LIN {X 0,Y 573.039,Z 679.467,A -85,B 0,C 180,E1 -2242.601,E2 -2242.601} C_VEL
LIN {X 0,Y 573.014,Z 684.186,A -85,B 0,C 180,E1 -2244.016,E2 -2244.016} C_VEL
LIN {X 0,Y 573.006,Z 688.636,A -85,B 0,C 180,E1 -2245.78,E2 -2245.78} C_VEL
LIN {X 0,Y 572.947,Z 691.089,A -85,B 0,C 180,E1 -2247.188,E2 -2247.188} C_VEL
LIN {X 0,Y 572.939,Z 692.479,A -85,B 0,C 180,E1 -2248.594,E2 -2248.594} C_VEL
LIN {X 0,Y 572.933,Z 693,A -85,B 0,C 180,E1 -2250,E2 -2250} C_VEL
LIN {X 0,Y 572.939,Z 692.479,A -85,B 0,C 180,E1 -2251.406,E2 -2251.406} C_VEL
LIN {X 0,Y 572.947,Z 691.088,A -85,B 0,C 180,E1 -2252.812,E2 -2252.812} C_VEL
LIN {X 0,Y 573.006,Z 688.635,A -85,B 0,C 180,E1 -2254.22,E2 -2254.22} C_VEL
LIN {X 0,Y 573.013,Z 684.187,A -85,B 0,C 180,E1 -2255.984,E2 -2255.984} C_VEL
LIN {X 0,Y 573.04,Z 679.468,A -85,B 0,C 180,E1 -2257.399,E2 -2257.399} C_VEL
LIN {X 0,Y 573.076,Z 673.488,A -85,B 0,C 180,E1 -2258.818,E2 -2258.818} C_VEL
LIN {X 0,Y 573.182,Z 665.275,A -85,B 0,C 180,E1 -2260.42,E2 -2260.42} C_VEL
LIN {X 0,Y 573.269,Z 656.443,A -85,B 0,C 180,E1 -2261.85,E2 -2261.85} C_VEL
LIN {X 0,Y 573.448,Z 645.907,A -85,B 0,C 180,E1 -2263.285,E2 -2263.285} C_VEL
LIN {X 0,Y 573.59,Z 635.033,A -85,B 0,C 180,E1 -2264.544,E2 -2264.544} C_VEL
LIN {X 0,Y 573.831,Z 624.069,A -85,B 0,C 180,E1 -2265.631,E2 -2265.631} C_VEL
LIN {X 0,Y 574.091,Z 610.219,A -85,B 0,C 180,E1 -2266.811,E2 -2266.811} C_VEL
LIN {X 0,Y 574.357,Z 596.263,A -85,B 0,C 180,E1 -2267.813,E2 -2267.813} C_VEL
LIN {X 0,Y 574.633,Z 582.712,A -85,B 0,C 180,E1 -2268.634,E2 -2268.634} C_VEL
LIN {X 0,Y 574.868,Z 568.146,A -85,B 0,C 180,E1 -2269.364,E2 -2269.364} C_VEL
LIN {X 0,Y 575.126,Z 552.237,A -85,B 0,C 180,E1 -2270.009,E2 -2270.009} C_VEL
LIN {X 0,Y 575.36,Z 536.004,A -85,B 0,C 180,E1 -2270.513,E2 -2270.513} C_VEL
LIN {X 0,Y 575.491,Z 519.421,A -85,B 0,C 180,E1 -2270.882,E2 -2270.882} C_VEL
LIN {X 0,Y 576.17,Z 335.886,A -85,B 0,C 180,E1 -2273.297,E2 -2273.297} C_VEL
LIN {X 0,Y 576.126,Z 317.819,A -85,B 0,C 180,E1 -2273.539,E2 -2273.539} C_VEL
LIN {X 0,Y 575.046,Z 311.756,A -85,B 0,C 180,E1 -2273.688,E2 -2273.688} C_VEL
LIN {X 0,Y 575.605,Z 275.985,A -85,B 0,C 180,E1 -2276.796,E2 -2276.796} C_VEL
LIN {X 0,Y 575.436,Z 270.86,A -85,B 0,C 180,E1 -2277.258,E2 -2277.258} C_VEL
LIN {X 0,Y 573.251,Z 263.391,A -85,B 0,C 180,E1 -2278.039,E2 -2278.039} C_VEL
LIN {X 0,Y 573.232,Z 263.394,A -85,B 0,C 180,E1 -2280.883,E2 -2280.883} C_VEL
LIN {X 0,Y 573.262,Z 263.391,A -85,B 0,C 180,E1 -2283.524,E2 -2283.524} C_VEL
LIN {X 0,Y 573.213,Z 263.391,A -85,B 0,C 180,E1 -2286.052,E2 -2286.052} C_VEL
LIN {X 0,Y 573.248,Z 263.39,A -85,B 0,C 180,E1 -2288.701,E2 -2288.701} C_VEL
LIN {X 0,Y 573.244,Z 263.388,A -85,B 0,C 180,E1 -2291.595,E2 -2291.595} C_VEL
LIN {X 0,Y 573.24,Z 263.388,A -85,B 0,C 180,E1 -2294.333,E2 -2294.333} C_VEL
LIN {X 0,Y 573.241,Z 263.391,A -85,B 0,C 180,E1 -2297.359,E2 -2297.359} C_VEL
LIN {X 0,Y 573.248,Z 263.387,A -85,B 0,C 180,E1 -2300.393,E2 -2300.393} C_VEL
LIN {X 0,Y 573.253,Z 263.393,A -85,B 0,C 180,E1 -2303.078,E2 -2303.078} C_VEL
LIN {X 0,Y 573.267,Z 263.383,A -85,B 0,C 180,E1 -2305.672,E2 -2305.672} C_VEL
LIN {X 0,Y 573.243,Z 263.386,A -85,B 0,C 180,E1 -2308.185,E2 -2308.185} C_VEL
LIN {X 0,Y 573.265,Z 263.39,A -85,B 0,C 180,E1 -2310.635,E2 -2310.635} C_VEL
LIN {X 0,Y 573.251,Z 263.392,A -85,B 0,C 180,E1 -2313.024,E2 -2313.024} C_VEL
LIN {X 0,Y 573.276,Z 263.383,A -85,B 0,C 180,E1 -2315.367,E2 -2315.367} C_VEL
LIN {X 0,Y 573.229,Z 263.39,A -85,B 0,C 180,E1 -2318.42,E2 -2318.42} C_VEL
LIN {X 0,Y 573.271,Z 263.392,A -85,B 0,C 180,E1 -2320.732,E2 -2320.732} C_VEL
LIN {X 0,Y 573.242,Z 263.383,A -85,B 0,C 180,E1 -2323.622,E2 -2323.622} C_VEL
LIN {X 0,Y 573.229,Z 263.396,A -85,B 0,C 180,E1 -2326.53,E2 -2326.53} C_VEL
LIN {X 0,Y 573.265,Z 263.387,A -85,B 0,C 180,E1 -2328.746,E2 -2328.746} C_VEL
LIN {X 0,Y 573.254,Z 263.385,A -85,B 0,C 180,E1 -2331.54,E2 -2331.54} C_VEL
LIN {X 0,Y 573.285,Z 263.388,A -85,B 0,C 180,E1 -2334.372,E2 -2334.372} C_VEL
LIN {X 0,Y 573.311,Z 263.379,A -85,B 0,C 180,E1 -2337.893,E2 -2337.893} C_VEL
LIN {X 0,Y 573.327,Z 263.379,A -85,B 0,C 180,E1 -2340.703,E2 -2340.703} C_VEL
LIN {X 0,Y 573.291,Z 263.383,A -85,B 0,C 180,E1 -2342.811,E2 -2342.811} C_VEL
LIN {X 0,Y 573.271,Z 263.384,A -85,B 0,C 180,E1 -2345.629,E2 -2345.629} C_VEL
LIN {X 0,Y 573.25,Z 263.392,A -85,B 0,C 180,E1 -2348.46,E2 -2348.46} C_VEL
LIN {X 0,Y 573.275,Z 263.382,A -85,B 0,C 180,E1 -2351.312,E2 -2351.312} C_VEL
LIN {X 0,Y 573.273,Z 263.389,A -85,B 0,C 180,E1 -2354.42,E2 -2354.42} C_VEL
LIN {X 0,Y 573.195,Z 263.392,A -85,B 0,C 180,E1 -2357.114,E2 -2357.114} C_VEL
LIN {X 0,Y 573.268,Z 263.38,A -85,B 0,C 180,E1 -2359.33,E2 -2359.33} C_VEL
LIN {X 0,Y 573.209,Z 263.396,A -85,B 0,C 180,E1 -2362.339,E2 -2362.339} C_VEL
LIN {X 0,Y 573.202,Z 263.393,A -85,B 0,C 180,E1 -2364.375,E2 -2364.375} C_VEL
LIN {X 0,Y 572.56,Z 263.474,A -85,B 0,C 180,E1 -2364.962,E2 -2364.962} C_VEL
LIN {X 0,Y 569.719,Z 263.832,A -85,B 0,C 180,E1 -2365.913,E2 -2365.913} C_VEL
LIN {X 0,Y 567.293,Z 264.131,A -85,B 0,C 180,E1 -2366.679,E2 -2366.679} C_VEL
LIN {X 0,Y 566.236,Z 264.26,A -85,B 0,C 180,E1 -2367.27,E2 -2367.27} C_VEL
LIN {X 0,Y 566.142,Z 264.271,A -85,B 0,C 180,E1 -2367.47,E2 -2367.47} C_VEL
LIN {X 0,Y 566.158,Z 264.271,A -85,B 0,C 180,E1 -2370.595,E2 -2370.595} C_VEL
LIN {X 0,Y 566.162,Z 264.269,A -85,B 0,C 180,E1 -2373.107,E2 -2373.107} C_VEL
LIN {X 0,Y 566.133,Z 264.277,A -85,B 0,C 180,E1 -2375.695,E2 -2375.695} C_VEL
LIN {X 0,Y 566.187,Z 264.267,A -85,B 0,C 180,E1 -2378.555,E2 -2378.555} C_VEL
LIN {X 0,Y 566.136,Z 264.272,A -85,B 0,C 180,E1 -2381.144,E2 -2381.144} C_VEL
LIN {X 0,Y 566.149,Z 264.278,A -85,B 0,C 180,E1 -2384.041,E2 -2384.041} C_VEL
LIN {X 0,Y 566.155,Z 264.271,A -85,B 0,C 180,E1 -2387.089,E2 -2387.089} C_VEL
LIN {X 0,Y 566.19,Z 264.272,A -85,B 0,C 180,E1 -2390.318,E2 -2390.318} C_VEL
LIN {X 0,Y 566.221,Z 264.448,A -85,B 0,C 180,E1 -2391.127,E2 -2391.127} C_VEL
LIN {X 0,Y 568.077,Z 271.603,A -85,B 0,C 180,E1 -2391.953,E2 -2391.953} C_VEL
LIN {X 0,Y 568.103,Z 283.142,A -85,B 0,C 180,E1 -2393.09,E2 -2393.09} C_VEL
LIN {X 0,Y 569.669,Z 290.812,A -85,B 0,C 180,E1 -2393.263,E2 -2393.263} C_VEL
LIN {X 0,Y 568.911,Z 488.882,A -85,B 0,C 180,E1 -2395.901,E2 -2395.901} C_VEL
LIN {X 0,Y 568.673,Z 505.398,A -85,B 0,C 180,E1 -2396.264,E2 -2396.264} C_VEL
LIN {X 0,Y 568.446,Z 520.462,A -85,B 0,C 180,E1 -2396.727,E2 -2396.727} C_VEL
LIN {X 0,Y 568.229,Z 534.795,A -85,B 0,C 180,E1 -2397.288,E2 -2397.288} C_VEL
LIN {X 0,Y 567.885,Z 550.466,A -85,B 0,C 180,E1 -2398.058,E2 -2398.058} C_VEL
LIN {X 0,Y 567.583,Z 565.698,A -85,B 0,C 180,E1 -2398.975,E2 -2398.975} C_VEL
LIN {X 0,Y 567.236,Z 579.436,A -85,B 0,C 180,E1 -2399.963,E2 -2399.963} C_VEL
LIN {X 0,Y 566.924,Z 592.685,A -85,B 0,C 180,E1 -2401.087,E2 -2401.087} C_VEL
LIN {X 0,Y 566.675,Z 604.723,A -85,B 0,C 180,E1 -2402.284,E2 -2402.284} C_VEL
LIN {X 0,Y 566.438,Z 616.523,A -85,B 0,C 180,E1 -2403.668,E2 -2403.668} C_VEL
LIN {X 0,Y 566.25,Z 626.398,A -85,B 0,C 180,E1 -2405.04,E2 -2405.04} C_VEL
LIN {X 0,Y 566.132,Z 634.748,A -85,B 0,C 180,E1 -2406.4,E2 -2406.4} C_VEL
LIN {X 0,Y 566.023,Z 641.81,A -85,B 0,C 180,E1 -2407.747,E2 -2407.747} C_VEL
LIN {X 0,Y 565.958,Z 648.363,A -85,B 0,C 180,E1 -2409.273,E2 -2409.273} C_VEL
LIN {X 0,Y 565.919,Z 653.355,A -85,B 0,C 180,E1 -2410.706,E2 -2410.706} C_VEL
LIN {X 0,Y 565.856,Z 656.694,A -85,B 0,C 180,E1 -2411.91,E2 -2411.91} C_VEL
LIN {X 0,Y 565.845,Z 659.849,A -85,B 0,C 180,E1 -2413.401,E2 -2413.401} C_VEL
LIN {X 0,Y 565.805,Z 661.86,A -85,B 0,C 180,E1 -2414.88,E2 -2414.88} C_VEL
LIN {X 0,Y 565.863,Z 662.853,A -85,B 0,C 180,E1 -2416.351,E2 -2416.351} C_VEL
LIN {X 0,Y 565.864,Z 662.837,A -85,B 0,C 180,E1 -2417.811,E2 -2417.811} C_VEL
LIN {X 0,Y 565.893,Z 661.802,A -85,B 0,C 180,E1 -2419.264,E2 -2419.264} C_VEL
LIN {X 0,Y 565.829,Z 659.82,A -85,B 0,C 180,E1 -2420.708,E2 -2420.708} C_VEL
LIN {X 0,Y 565.879,Z 656.772,A -85,B 0,C 180,E1 -2422.148,E2 -2422.148} C_VEL
LIN {X 0,Y 565.948,Z 652.76,A -85,B 0,C 180,E1 -2423.583,E2 -2423.583} C_VEL
LIN {X 0,Y 565.989,Z 646.166,A -85,B 0,C 180,E1 -2425.37,E2 -2425.37} C_VEL
LIN {X 0,Y 566.057,Z 639.533,A -85,B 0,C 180,E1 -2426.797,E2 -2426.797} C_VEL
LIN {X 0,Y 566.173,Z 630.559,A -85,B 0,C 180,E1 -2428.399,E2 -2428.399} C_VEL
LIN {X 0,Y 566.305,Z 621.025,A -85,B 0,C 180,E1 -2429.822,E2 -2429.822} C_VEL
LIN {X 0,Y 566.52,Z 609.741,A -85,B 0,C 180,E1 -2431.244,E2 -2431.244} C_VEL
LIN {X 0,Y 566.818,Z 598.124,A -85,B 0,C 180,E1 -2432.487,E2 -2432.487} C_VEL
LIN {X 0,Y 567.115,Z 585.432,A -85,B 0,C 180,E1 -2433.641,E2 -2433.641} C_VEL
LIN {X 0,Y 567.384,Z 571.676,A -85,B 0,C 180,E1 -2434.707,E2 -2434.707} C_VEL
LIN {X 0,Y 567.697,Z 556.622,A -85,B 0,C 180,E1 -2435.684,E2 -2435.684} C_VEL
LIN {X 0,Y 568.054,Z 541.711,A -85,B 0,C 180,E1 -2436.482,E2 -2436.482} C_VEL
LIN {X 0,Y 568.372,Z 526.427,A -85,B 0,C 180,E1 -2437.147,E2 -2437.147} C_VEL
LIN {X 0,Y 568.633,Z 509.883,A -85,B 0,C 180,E1 -2437.702,E2 -2437.702} C_VEL
LIN {X 0,Y 568.827,Z 493.69,A -85,B 0,C 180,E1 -2438.096,E2 -2438.096} C_VEL
LIN {X 0,Y 568.984,Z 472.324,A -85,B 0,C 180,E1 -2438.426,E2 -2438.426} C_VEL
LIN {X 0,Y 569.662,Z 291.209,A -85,B 0,C 180,E1 -2440.822,E2 -2440.822} C_VEL
LIN {X 0,Y 568.055,Z 282.844,A -85,B 0,C 180,E1 -2441.011,E2 -2441.011} C_VEL
LIN {X 0,Y 568.099,Z 271.56,A -85,B 0,C 180,E1 -2442.14,E2 -2442.14} C_VEL
LIN {X 0,Y 566.179,Z 264.273,A -85,B 0,C 180,E1 -2443.002,E2 -2443.002} C_VEL
LIN {X 0,Y 566.189,Z 264.268,A -85,B 0,C 180,E1 -2445.11,E2 -2445.11} C_VEL
LIN {X 0,Y 566.171,Z 264.275,A -85,B 0,C 180,E1 -2448.079,E2 -2448.079} C_VEL
LIN {X 0,Y 566.197,Z 264.273,A -85,B 0,C 180,E1 -2450.338,E2 -2450.338} C_VEL
LIN {X 0,Y 566.17,Z 264.269,A -85,B 0,C 180,E1 -2453.28,E2 -2453.28} C_VEL
LIN {X 0,Y 566.174,Z 264.27,A -85,B 0,C 180,E1 -2455.751,E2 -2455.751} C_VEL
LIN {X 0,Y 566.138,Z 264.282,A -85,B 0,C 180,E1 -2458.189,E2 -2458.189} C_VEL
LIN {X 0,Y 566.176,Z 264.267,A -85,B 0,C 180,E1 -2461.073,E2 -2461.073} C_VEL
LIN {X 0,Y 566.184,Z 264.274,A -85,B 0,C 180,E1 -2463.958,E2 -2463.958} C_VEL
LIN {X 0,Y 566.122,Z 264.276,A -85,B 0,C 180,E1 -2466.576,E2 -2466.576} C_VEL
LIN {X 0,Y 566.179,Z 264.27,A -85,B 0,C 180,E1 -2469.681,E2 -2469.681} C_VEL
LIN {X 0,Y 566.144,Z 264.27,A -85,B 0,C 180,E1 -2472.91,E2 -2472.91} C_VEL
LIN {X 0,Y 566.146,Z 264.278,A -85,B 0,C 180,E1 -2475.959,E2 -2475.959} C_VEL
LIN {X 0,Y 566.135,Z 264.272,A -85,B 0,C 180,E1 -2478.856,E2 -2478.856} C_VEL
LIN {X 0,Y 566.174,Z 264.271,A -85,B 0,C 180,E1 -2481.635,E2 -2481.635} C_VEL
LIN {X 0,Y 566.136,Z 264.27,A -85,B 0,C 180,E1 -2484.305,E2 -2484.305} C_VEL
LIN {X 0,Y 566.164,Z 264.267,A -85,B 0,C 180,E1 -2486.894,E2 -2486.894} C_VEL
LIN {X 0,Y 566.168,Z 264.272,A -85,B 0,C 180,E1 -2489.406,E2 -2489.406} C_VEL
LIN {X 0,Y 566.144,Z 264.279,A -85,B 0,C 180,E1 -2491.853,E2 -2491.853} C_VEL
LIN {X 0,Y 566.185,Z 264.267,A -85,B 0,C 180,E1 -2494.249,E2 -2494.249} C_VEL
LIN {X 0,Y 566.168,Z 264.265,A -85,B 0,C 180,E1 -2496.72,E2 -2496.72} C_VEL
LIN {X 0,Y 566.204,Z 264.273,A -85,B 0,C 180,E1 -2499.662,E2 -2499.662} C_VEL
LIN {X 0,Y 566.18,Z 264.269,A -85,B 0,C 180,E1 -2501.921,E2 -2501.921} C_VEL
LIN {X 0,Y 566.19,Z 264.266,A -85,B 0,C 180,E1 -2504.89,E2 -2504.89} C_VEL
LIN {X 0,Y 566.217,Z 264.265,A -85,B 0,C 180,E1 -2507.818,E2 -2507.818} C_VEL
LIN {X 0,Y 566.17,Z 264.27,A -85,B 0,C 180,E1 -2509.992,E2 -2509.992} C_VEL
LIN {X 0,Y 566.237,Z 264.26,A -85,B 0,C 180,E1 -2512.87,E2 -2512.87} C_VEL
LIN {X 0,Y 566.274,Z 264.255,A -85,B 0,C 180,E1 -2515.016,E2 -2515.016} C_VEL
LIN {X 0,Y 566.284,Z 264.256,A -85,B 0,C 180,E1 -2517.866,E2 -2517.866} C_VEL
LIN {X 0,Y 566.292,Z 264.25,A -85,B 0,C 180,E1 -2520.711,E2 -2520.711} C_VEL
LIN {X 0,Y 566.263,Z 264.258,A -85,B 0,C 180,E1 -2522.845,E2 -2522.845} C_VEL
LIN {X 0,Y 566.263,Z 264.257,A -85,B 0,C 180,E1 -2525.698,E2 -2525.698} C_VEL
LIN {X 0,Y 566.226,Z 264.259,A -85,B 0,C 180,E1 -2528.565,E2 -2528.565} C_VEL
LIN {X 0,Y 566.243,Z 264.265,A -85,B 0,C 180,E1 -2531.454,E2 -2531.454} C_VEL
LIN {X 0,Y 566.224,Z 264.262,A -85,B 0,C 180,E1 -2534.502,E2 -2534.502} C_VEL
LIN {X 0,Y 566.2,Z 264.272,A -85,B 0,C 180,E1 -2537.331,E2 -2537.331} C_VEL
LIN {X 0,Y 566.207,Z 264.263,A -85,B 0,C 180,E1 -2540.337,E2 -2540.337} C_VEL
LIN {X 0,Y 566.19,Z 264.271,A -85,B 0,C 180,E1 -2543.403,E2 -2543.403} C_VEL
LIN {X 0,Y 566.213,Z 264.264,A -85,B 0,C 180,E1 -2545.749,E2 -2545.749} C_VEL
LIN {X 0,Y 566.202,Z 264.263,A -85,B 0,C 180,E1 -2548.202,E2 -2548.202} C_VEL
LIN {X 0,Y 566.191,Z 264.274,A -85,B 0,C 180,E1 -2551.076,E2 -2551.076} C_VEL
LIN {X 0,Y 566.211,Z 264.263,A -85,B 0,C 180,E1 -2553.734,E2 -2553.734} C_VEL
LIN {X 0,Y 566.209,Z 264.265,A -85,B 0,C 180,E1 -2556.569,E2 -2556.569} C_VEL
LIN {X 0,Y 566.212,Z 264.263,A -85,B 0,C 180,E1 -2559.685,E2 -2559.685} C_VEL
LIN {X 0,Y 566.21,Z 264.263,A -85,B 0,C 180,E1 -2562.087,E2 -2562.087} C_VEL
LIN {X 0,Y 566.173,Z 264.275,A -85,B 0,C 180,E1 -2565.036,E2 -2565.036} C_VEL
LIN {X 0,Y 566.217,Z 264.262,A -85,B 0,C 180,E1 -2568.136,E2 -2568.136} C_VEL
LIN {X 0,Y 566.22,Z 264.271,A -85,B 0,C 180,E1 -2570.727,E2 -2570.727} C_VEL
LIN {X 0,Y 566.184,Z 264.266,A -85,B 0,C 180,E1 -2573.788,E2 -2573.788} C_VEL
LIN {X 0,Y 566.21,Z 264.266,A -85,B 0,C 180,E1 -2576.266,E2 -2576.266} C_VEL
LIN {X 0,Y 566.192,Z 264.273,A -85,B 0,C 180,E1 -2578.923,E2 -2578.923} C_VEL
LIN {X 0,Y 566.241,Z 264.43,A -85,B 0,C 180,E1 -2581.703,E2 -2581.703} C_VEL
LIN {X 0,Y 568.802,Z 273.142,A -85,B 0,C 180,E1 -2582.617,E2 -2582.617} C_VEL
LIN {X 0,Y 568.734,Z 288.517,A -85,B 0,C 180,E1 -2583.98,E2 -2583.98} C_VEL
LIN {X 0,Y 568.339,Z 311.989,A -85,B 0,C 180,E1 -2586.035,E2 -2586.035} C_VEL
LIN {X 0,Y 569.734,Z 319.826,A -85,B 0,C 180,E1 -2586.208,E2 -2586.208} C_VEL
LIN {X 0,Y 568.878,Z 519.43,A -85,B 0,C 180,E1 -2588.864,E2 -2588.864} C_VEL
LIN {X 0,Y 568.726,Z 536.008,A -85,B 0,C 180,E1 -2589.237,E2 -2589.237} C_VEL
LIN {X 0,Y 568.422,Z 552.242,A -85,B 0,C 180,E1 -2589.745,E2 -2589.745} C_VEL
LIN {X 0,Y 568.145,Z 568.386,A -85,B 0,C 180,E1 -2590.408,E2 -2590.408} C_VEL
LIN {X 0,Y 567.878,Z 582.716,A -85,B 0,C 180,E1 -2591.136,E2 -2591.136} C_VEL
LIN {X 0,Y 567.582,Z 596.269,A -85,B 0,C 180,E1 -2591.967,E2 -2591.967} C_VEL
LIN {X 0,Y 567.228,Z 610.219,A -85,B 0,C 180,E1 -2592.979,E2 -2592.979} C_VEL
LIN {X 0,Y 566.915,Z 624.07,A -85,B 0,C 180,E1 -2594.173,E2 -2594.173} C_VEL
LIN {X 0,Y 566.63,Z 635.619,A -85,B 0,C 180,E1 -2595.339,E2 -2595.339} C_VEL
LIN {X 0,Y 566.434,Z 647.337,A -85,B 0,C 180,E1 -2596.73,E2 -2596.73} C_VEL
LIN {X 0,Y 566.238,Z 657.673,A -85,B 0,C 180,E1 -2598.183,E2 -2598.183} C_VEL
LIN {X 0,Y 566.12,Z 666.284,A -85,B 0,C 180,E1 -2599.63,E2 -2599.63} C_VEL
LIN {X 0,Y 566.001,Z 673.489,A -85,B 0,C 180,E1 -2601.071,E2 -2601.071} C_VEL
LIN {X 0,Y 565.968,Z 679.467,A -85,B 0,C 180,E1 -2602.508,E2 -2602.508} C_VEL
LIN {X 0,Y 565.915,Z 684.187,A -85,B 0,C 180,E1 -2603.941,E2 -2603.941} C_VEL
LIN {X 0,Y 565.911,Z 688.637,A -85,B 0,C 180,E1 -2605.727,E2 -2605.727} C_VEL
LIN {X 0,Y 565.865,Z 691.089,A -85,B 0,C 180,E1 -2607.152,E2 -2607.152} C_VEL
LIN {X 0,Y 565.839,Z 692.48,A -85,B 0,C 180,E1 -2608.577,E2 -2608.577} C_VEL
LIN {X 0,Y 565.834,Z 693,A -85,B 0,C 180,E1 -2610,E2 -2610} C_VEL
LIN {X 0,Y 565.839,Z 692.48,A -85,B 0,C 180,E1 -2611.424,E2 -2611.424} C_VEL
LIN {X 0,Y 565.866,Z 691.088,A -85,B 0,C 180,E1 -2612.848,E2 -2612.848} C_VEL
LIN {X 0,Y 565.911,Z 688.636,A -85,B 0,C 180,E1 -2614.273,E2 -2614.273} C_VEL
LIN {X 0,Y 565.914,Z 684.188,A -85,B 0,C 180,E1 -2616.06,E2 -2616.06} C_VEL
LIN {X 0,Y 565.968,Z 679.468,A -85,B 0,C 180,E1 -2617.492,E2 -2617.492} C_VEL
LIN {X 0,Y 566.001,Z 673.489,A -85,B 0,C 180,E1 -2618.929,E2 -2618.929} C_VEL
LIN {X 0,Y 566.126,Z 665.276,A -85,B 0,C 180,E1 -2620.551,E2 -2620.551} C_VEL
LIN {X 0,Y 566.246,Z 656.442,A -85,B 0,C 180,E1 -2621.999,E2 -2621.999} C_VEL
LIN {X 0,Y 566.427,Z 645.907,A -85,B 0,C 180,E1 -2623.453,E2 -2623.453} C_VEL
LIN {X 0,Y 566.661,Z 634.61,A -85,B 0,C 180,E1 -2624.774,E2 -2624.774} C_VEL
LIN {X 0,Y 566.958,Z 622.117,A -85,B 0,C 180,E1 -2626.01,E2 -2626.01} C_VEL
LIN {X 0,Y 567.229,Z 609.043,A -85,B 0,C 180,E1 -2627.113,E2 -2627.113} C_VEL
LIN {X 0,Y 567.581,Z 594.848,A -85,B 0,C 180,E1 -2628.126,E2 -2628.126} C_VEL
LIN {X 0,Y 567.907,Z 579.276,A -85,B 0,C 180,E1 -2629.05,E2 -2629.05} C_VEL
LIN {X 0,Y 568.272,Z 563.648,A -85,B 0,C 180,E1 -2629.804,E2 -2629.804} C_VEL
LIN {X 0,Y 568.551,Z 547.003,A -85,B 0,C 180,E1 -2630.439,E2 -2630.439} C_VEL
LIN {X 0,Y 568.778,Z 530.512,A -85,B 0,C 180,E1 -2630.903,E2 -2630.903} C_VEL
LIN {X 0,Y 568.899,Z 514.918,A -85,B 0,C 180,E1 -2631.207,E2 -2631.207} C_VEL
LIN {X 0,Y 569.679,Z 320,A -85,B 0,C 180,E1 -2633.792,E2 -2633.792} C_VEL
LIN {X 0,Y 568.354,Z 311.822,A -85,B 0,C 180,E1 -2633.979,E2 -2633.979} C_VEL
LIN {X 0,Y 568.944,Z 276.843,A -85,B 0,C 180,E1 -2637.044,E2 -2637.044} C_VEL
LIN {X 0,Y 568.742,Z 272.884,A -85,B 0,C 180,E1 -2637.406,E2 -2637.406} C_VEL
LIN {X 0,Y 566.216,Z 264.268,A -85,B 0,C 180,E1 -2638.324,E2 -2638.324} C_VEL
LIN {X 0,Y 566.195,Z 264.273,A -85,B 0,C 180,E1 -2641.422,E2 -2641.422} C_VEL
LIN {X 0,Y 566.209,Z 264.265,A -85,B 0,C 180,E1 -2643.956,E2 -2643.956} C_VEL
LIN {X 0,Y 566.199,Z 264.267,A -85,B 0,C 180,E1 -2646.57,E2 -2646.57} C_VEL
LIN {X 0,Y 566.221,Z 264.269,A -85,B 0,C 180,E1 -2649.273,E2 -2649.273} C_VEL
LIN {X 0,Y 566.211,Z 264.261,A -85,B 0,C 180,E1 -2652.088,E2 -2652.088} C_VEL
LIN {X 0,Y 566.174,Z 264.274,A -85,B 0,C 180,E1 -2655.036,E2 -2655.036} C_VEL
LIN {X 0,Y 566.218,Z 264.261,A -85,B 0,C 180,E1 -2658.136,E2 -2658.136} C_VEL
LIN {X 0,Y 566.223,Z 264.267,A -85,B 0,C 180,E1 -2660.727,E2 -2660.727} C_VEL
LIN {X 0,Y 566.185,Z 264.266,A -85,B 0,C 180,E1 -2663.788,E2 -2663.788} C_VEL
LIN {X 0,Y 566.212,Z 264.263,A -85,B 0,C 180,E1 -2666.266,E2 -2666.266} C_VEL
LIN {X 0,Y 566.194,Z 264.274,A -85,B 0,C 180,E1 -2668.924,E2 -2668.924} C_VEL
LIN {X 0,Y 566.213,Z 264.258,A -85,B 0,C 180,E1 -2671.858,E2 -2671.858} C_VEL
LIN {X 0,Y 566.214,Z 264.264,A -85,B 0,C 180,E1 -2674.251,E2 -2674.251} C_VEL
LIN {X 0,Y 566.174,Z 264.273,A -85,B 0,C 180,E1 -2676.719,E2 -2676.719} C_VEL
LIN {X 0,Y 566.207,Z 264.263,A -85,B 0,C 180,E1 -2679.663,E2 -2679.663} C_VEL
LIN {X 0,Y 566.201,Z 264.268,A -85,B 0,C 180,E1 -2682.669,E2 -2682.669} C_VEL
LIN {X 0,Y 566.223,Z 264.261,A -85,B 0,C 180,E1 -2685.627,E2 -2685.627} C_VEL
LIN {X 0,Y 566.237,Z 264.263,A -85,B 0,C 180,E1 -2688.676,E2 -2688.676} C_VEL
LIN {X 0,Y 566.205,Z 264.263,A -85,B 0,C 180,E1 -2691.434,E2 -2691.434} C_VEL
LIN {X 0,Y 566.253,Z 264.263,A -85,B 0,C 180,E1 -2694.302,E2 -2694.302} C_VEL
LIN {X 0,Y 566.282,Z 264.254,A -85,B 0,C 180,E1 -2697.867,E2 -2697.867} C_VEL
LIN {X 0,Y 566.298,Z 264.253,A -85,B 0,C 180,E1 -2700.711,E2 -2700.711} C_VEL
LIN {X 0,Y 566.257,Z 264.259,A -85,B 0,C 180,E1 -2702.846,E2 -2702.846} C_VEL
LIN {X 0,Y 566.241,Z 264.26,A -85,B 0,C 180,E1 -2705.699,E2 -2705.699} C_VEL
LIN {X 0,Y 566.201,Z 264.268,A -85,B 0,C 180,E1 -2708.567,E2 -2708.567} C_VEL
LIN {X 0,Y 566.243,Z 264.259,A -85,B 0,C 180,E1 -2711.455,E2 -2711.455} C_VEL
LIN {X 0,Y 566.227,Z 264.265,A -85,B 0,C 180,E1 -2714.502,E2 -2714.502} C_VEL
LIN {X 0,Y 566.161,Z 264.269,A -85,B 0,C 180,E1 -2717.333,E2 -2717.333} C_VEL
LIN {X 0,Y 566.199,Z 264.261,A -85,B 0,C 180,E1 -2719.581,E2 -2719.581} C_VEL
LIN {X 0,Y 566.179,Z 264.272,A -85,B 0,C 180,E1 -2721.864,E2 -2721.864} C_VEL
LIN {X 0,Y 566.15,Z 264.273,A -85,B 0,C 180,E1 -2724.372,E2 -2724.372} C_VEL
LIN {X 0,Y 566.16,Z 264.271,A -85,B 0,C 180,E1 -2726.649,E2 -2726.649} C_VEL
LIN {X 0,Y 566.142,Z 264.271,A -85,B 0,C 180,E1 -2727.47,E2 -2727.47} C_VEL
LIN {X 0,Y 565.452,Z 264.363,A -85,B 0,C 180,E1 -2728.064,E2 -2728.064} C_VEL
LIN {X 0,Y 562.584,Z 264.72,A -85,B 0,C 180,E1 -2729.028,E2 -2729.028} C_VEL
LIN {X 0,Y 560.187,Z 265.019,A -85,B 0,C 180,E1 -2729.803,E2 -2729.803} C_VEL
LIN {X 0,Y 559.177,Z 265.144,A -85,B 0,C 180,E1 -2730.402,E2 -2730.402} C_VEL
LIN {X 0,Y 559.105,Z 265.15,A -85,B 0,C 180,E1 -2730.605,E2 -2730.605} C_VEL
LIN {X 0,Y 559.134,Z 265.145,A -85,B 0,C 180,E1 -2732.717,E2 -2732.717} C_VEL
LIN {X 0,Y 559.111,Z 265.148,A -85,B 0,C 180,E1 -2735.326,E2 -2735.326} C_VEL
LIN {X 0,Y 559.108,Z 265.154,A -85,B 0,C 180,E1 -2738.02,E2 -2738.02} C_VEL
LIN {X 0,Y 559.093,Z 265.149,A -85,B 0,C 180,E1 -2740.819,E2 -2740.819} C_VEL
LIN {X 0,Y 559.095,Z 265.158,A -85,B 0,C 180,E1 -2743.739,E2 -2743.739} C_VEL
LIN {X 0,Y 559.103,Z 265.152,A -85,B 0,C 180,E1 -2746.262,E2 -2746.262} C_VEL
LIN {X 0,Y 559.098,Z 265.151,A -85,B 0,C 180,E1 -2748.958,E2 -2748.958} C_VEL
LIN {X 0,Y 559.192,Z 265.316,A -85,B 0,C 180,E1 -2750.847,E2 -2750.847} C_VEL
LIN {X 0,Y 561.485,Z 274.746,A -85,B 0,C 180,E1 -2751.943,E2 -2751.943} C_VEL
LIN {X 0,Y 561.415,Z 283.251,A -85,B 0,C 180,E1 -2752.786,E2 -2752.786} C_VEL
LIN {X 0,Y 563.161,Z 291.947,A -85,B 0,C 180,E1 -2752.986,E2 -2752.986} C_VEL
LIN {X 0,Y 562.3,Z 486.908,A -85,B 0,C 180,E1 -2755.609,E2 -2755.609} C_VEL
LIN {X 0,Y 562.049,Z 503.604,A -85,B 0,C 180,E1 -2755.961,E2 -2755.961} C_VEL
LIN {X 0,Y 561.792,Z 519.55,A -85,B 0,C 180,E1 -2756.442,E2 -2756.442} C_VEL
LIN {X 0,Y 561.511,Z 535.019,A -85,B 0,C 180,E1 -2757.051,E2 -2757.051} C_VEL
LIN {X 0,Y 561.106,Z 550.799,A -85,B 0,C 180,E1 -2757.837,E2 -2757.837} C_VEL
LIN {X 0,Y 560.784,Z 565.257,A -85,B 0,C 180,E1 -2758.719,E2 -2758.719} C_VEL
LIN {X 0,Y 560.394,Z 578.625,A -85,B 0,C 180,E1 -2759.683,E2 -2759.683} C_VEL
LIN {X 0,Y 560.049,Z 591.799,A -85,B 0,C 180,E1 -2760.801,E2 -2760.801} C_VEL
LIN {X 0,Y 559.724,Z 604.87,A -85,B 0,C 180,E1 -2762.114,E2 -2762.114} C_VEL
LIN {X 0,Y 559.444,Z 616.653,A -85,B 0,C 180,E1 -2763.515,E2 -2763.515} C_VEL
LIN {X 0,Y 559.231,Z 625.839,A -85,B 0,C 180,E1 -2764.803,E2 -2764.803} C_VEL
LIN {X 0,Y 559.07,Z 634.839,A -85,B 0,C 180,E1 -2766.28,E2 -2766.28} C_VEL
LIN {X 0,Y 558.93,Z 642.764,A -85,B 0,C 180,E1 -2767.838,E2 -2767.838} C_VEL
LIN {X 0,Y 558.857,Z 649.181,A -85,B 0,C 180,E1 -2769.383,E2 -2769.383} C_VEL
LIN {X 0,Y 558.814,Z 654.204,A -85,B 0,C 180,E1 -2770.914,E2 -2770.914} C_VEL
LIN {X 0,Y 558.756,Z 658.059,A -85,B 0,C 180,E1 -2772.43,E2 -2772.43} C_VEL
LIN {X 0,Y 558.728,Z 660.745,A -85,B 0,C 180,E1 -2773.935,E2 -2773.935} C_VEL
LIN {X 0,Y 558.763,Z 662.464,A -85,B 0,C 180,E1 -2775.58,E2 -2775.58} C_VEL
LIN {X 0,Y 558.741,Z 662.978,A -85,B 0,C 180,E1 -2776.914,E2 -2776.914} C_VEL
LIN {X 0,Y 558.801,Z 662.261,A -85,B 0,C 180,E1 -2778.816,E2 -2778.816} C_VEL
LIN {X 0,Y 558.778,Z 661.178,A -85,B 0,C 180,E1 -2779.858,E2 -2779.858} C_VEL
LIN {X 0,Y 558.766,Z 658.745,A -85,B 0,C 180,E1 -2781.319,E2 -2781.319} C_VEL
LIN {X 0,Y 558.804,Z 655.375,A -85,B 0,C 180,E1 -2782.775,E2 -2782.775} C_VEL
LIN {X 0,Y 558.87,Z 649.627,A -85,B 0,C 180,E1 -2784.588,E2 -2784.588} C_VEL
LIN {X 0,Y 558.954,Z 643.725,A -85,B 0,C 180,E1 -2786.035,E2 -2786.035} C_VEL
LIN {X 0,Y 559.022,Z 636.671,A -85,B 0,C 180,E1 -2787.478,E2 -2787.478} C_VEL
LIN {X 0,Y 559.198,Z 628.262,A -85,B 0,C 180,E1 -2788.92,E2 -2788.92} C_VEL
LIN {X 0,Y 559.336,Z 618.269,A -85,B 0,C 180,E1 -2790.36,E2 -2790.36} C_VEL
LIN {X 0,Y 559.601,Z 608.024,A -85,B 0,C 180,E1 -2791.619,E2 -2791.619} C_VEL
LIN {X 0,Y 559.941,Z 596.116,A -85,B 0,C 180,E1 -2792.878,E2 -2792.878} C_VEL
LIN {X 0,Y 560.32,Z 583.146,A -85,B 0,C 180,E1 -2794.046,E2 -2794.046} C_VEL
LIN {X 0,Y 560.596,Z 571.449,A -85,B 0,C 180,E1 -2794.944,E2 -2794.944} C_VEL
LIN {X 0,Y 560.876,Z 557.881,A -85,B 0,C 180,E1 -2795.843,E2 -2795.843} C_VEL
LIN {X 0,Y 561.289,Z 543.266,A -85,B 0,C 180,E1 -2796.651,E2 -2796.651} C_VEL
LIN {X 0,Y 561.657,Z 527.124,A -85,B 0,C 180,E1 -2797.369,E2 -2797.369} C_VEL
LIN {X 0,Y 561.961,Z 511.524,A -85,B 0,C 180,E1 -2797.907,E2 -2797.907} C_VEL
LIN {X 0,Y 562.215,Z 495.019,A -85,B 0,C 180,E1 -2798.328,E2 -2798.328} C_VEL
LIN {X 0,Y 562.362,Z 477.198,A -85,B 0,C 180,E1 -2798.625,E2 -2798.625} C_VEL
LIN {X 0,Y 563.153,Z 291.665,A -85,B 0,C 180,E1 -2801.108,E2 -2801.108} C_VEL
LIN {X 0,Y 561.326,Z 282.817,A -85,B 0,C 180,E1 -2801.327,E2 -2801.327} C_VEL
LIN {X 0,Y 561.356,Z 273.43,A -85,B 0,C 180,E1 -2802.288,E2 -2802.288} C_VEL
LIN {X 0,Y 559.162,Z 265.147,A -85,B 0,C 180,E1 -2803.284,E2 -2803.284} C_VEL
LIN {X 0,Y 559.137,Z 265.147,A -85,B 0,C 180,E1 -2805.305,E2 -2805.305} C_VEL
LIN {X 0,Y 559.125,Z 265.147,A -85,B 0,C 180,E1 -2807.558,E2 -2807.558} C_VEL
LIN {X 0,Y 559.164,Z 265.145,A -85,B 0,C 180,E1 -2809.838,E2 -2809.838} C_VEL
LIN {X 0,Y 559.132,Z 265.15,A -85,B 0,C 180,E1 -2812.153,E2 -2812.153} C_VEL
LIN {X 0,Y 559.141,Z 265.143,A -85,B 0,C 180,E1 -2815.177,E2 -2815.177} C_VEL
LIN {X 0,Y 559.098,Z 265.152,A -85,B 0,C 180,E1 -2817.717,E2 -2817.717} C_VEL
LIN {X 0,Y 559.13,Z 265.155,A -85,B 0,C 180,E1 -2820.184,E2 -2820.184} C_VEL
LIN {X 0,Y 559.135,Z 265.146,A -85,B 0,C 180,E1 -2822.717,E2 -2822.717} C_VEL
LIN {X 0,Y 559.112,Z 265.146,A -85,B 0,C 180,E1 -2825.325,E2 -2825.325} C_VEL
LIN {X 0,Y 559.085,Z 265.158,A -85,B 0,C 180,E1 -2828.021,E2 -2828.021} C_VEL
LIN {X 0,Y 559.119,Z 265.154,A -85,B 0,C 180,E1 -2829.936,E2 -2829.936} C_VEL
LIN {X 0,Y 559.108,Z 265.147,A -85,B 0,C 180,E1 -2832.748,E2 -2832.748} C_VEL
LIN {X 0,Y 559.114,Z 265.153,A -85,B 0,C 180,E1 -2835.765,E2 -2835.765} C_VEL
LIN {X 0,Y 559.095,Z 265.154,A -85,B 0,C 180,E1 -2838.223,E2 -2838.223} C_VEL
LIN {X 0,Y 559.168,Z 265.139,A -85,B 0,C 180,E1 -2841.193,E2 -2841.193} C_VEL
LIN {X 0,Y 559.108,Z 265.146,A -85,B 0,C 180,E1 -2843.786,E2 -2843.786} C_VEL
LIN {X 0,Y 559.138,Z 265.144,A -85,B 0,C 180,E1 -2846.423,E2 -2846.423} C_VEL
LIN {X 0,Y 559.149,Z 265.142,A -85,B 0,C 180,E1 -2848.98,E2 -2848.98} C_VEL
LIN {X 0,Y 559.105,Z 265.152,A -85,B 0,C 180,E1 -2851.631,E2 -2851.631} C_VEL
LIN {X 0,Y 559.126,Z 265.144,A -85,B 0,C 180,E1 -2854.699,E2 -2854.699} C_VEL
LIN {X 0,Y 559.119,Z 265.145,A -85,B 0,C 180,E1 -2857.066,E2 -2857.066} C_VEL
LIN {X 0,Y 559.175,Z 265.144,A -85,B 0,C 180,E1 -2859.395,E2 -2859.395} C_VEL
LIN {X 0,Y 559.129,Z 265.15,A -85,B 0,C 180,E1 -2861.685,E2 -2861.685} C_VEL
LIN {X 0,Y 559.145,Z 265.147,A -85,B 0,C 180,E1 -2863.947,E2 -2863.947} C_VEL
LIN {X 0,Y 559.16,Z 265.142,A -85,B 0,C 180,E1 -2866.183,E2 -2866.183} C_VEL
LIN {X 0,Y 559.193,Z 265.137,A -85,B 0,C 180,E1 -2869.133,E2 -2869.133} C_VEL
LIN {X 0,Y 559.173,Z 265.141,A -85,B 0,C 180,E1 -2872.053,E2 -2872.053} C_VEL
LIN {X 0,Y 559.248,Z 265.129,A -85,B 0,C 180,E1 -2874.953,E2 -2874.953} C_VEL
LIN {X 0,Y 559.255,Z 265.132,A -85,B 0,C 180,E1 -2877.839,E2 -2877.839} C_VEL
LIN {X 0,Y 559.264,Z 265.125,A -85,B 0,C 180,E1 -2880.72,E2 -2880.72} C_VEL
LIN {X 0,Y 559.231,Z 265.134,A -85,B 0,C 180,E1 -2882.881,E2 -2882.881} C_VEL
LIN {X 0,Y 559.231,Z 265.132,A -85,B 0,C 180,E1 -2885.77,E2 -2885.77} C_VEL
LIN {X 0,Y 559.185,Z 265.137,A -85,B 0,C 180,E1 -2888.674,E2 -2888.674} C_VEL
LIN {X 0,Y 559.206,Z 265.139,A -85,B 0,C 180,E1 -2891.6,E2 -2891.6} C_VEL
LIN {X 0,Y 559.181,Z 265.14,A -85,B 0,C 180,E1 -2894.587,E2 -2894.587} C_VEL
LIN {X 0,Y 559.143,Z 265.147,A -85,B 0,C 180,E1 -2897.557,E2 -2897.557} C_VEL
LIN {X 0,Y 559.166,Z 265.142,A -85,B 0,C 180,E1 -2899.837,E2 -2899.837} C_VEL
LIN {X 0,Y 559.141,Z 265.143,A -85,B 0,C 180,E1 -2902.152,E2 -2902.152} C_VEL
LIN {X 0,Y 559.179,Z 265.147,A -85,B 0,C 180,E1 -2905.187,E2 -2905.187} C_VEL
LIN {X 0,Y 559.157,Z 265.142,A -85,B 0,C 180,E1 -2907.713,E2 -2907.713} C_VEL
LIN {X 0,Y 559.153,Z 265.142,A -85,B 0,C 180,E1 -2910.182,E2 -2910.182} C_VEL
LIN {X 0,Y 559.156,Z 265.147,A -85,B 0,C 180,E1 -2912.715,E2 -2912.715} C_VEL
LIN {X 0,Y 559.144,Z 265.146,A -85,B 0,C 180,E1 -2915.322,E2 -2915.322} C_VEL
LIN {X 0,Y 559.135,Z 265.144,A -85,B 0,C 180,E1 -2918.017,E2 -2918.017} C_VEL
LIN {X 0,Y 559.175,Z 265.146,A -85,B 0,C 180,E1 -2920.81,E2 -2920.81} C_VEL
LIN {X 0,Y 559.14,Z 265.143,A -85,B 0,C 180,E1 -2923.734,E2 -2923.734} C_VEL
LIN {X 0,Y 559.167,Z 265.149,A -85,B 0,C 180,E1 -2926.801,E2 -2926.801} C_VEL
LIN {X 0,Y 559.176,Z 265.144,A -85,B 0,C 180,E1 -2929.189,E2 -2929.189} C_VEL
LIN {X 0,Y 559.133,Z 265.145,A -85,B 0,C 180,E1 -2931.982,E2 -2931.982} C_VEL
LIN {X 0,Y 559.13,Z 265.152,A -85,B 0,C 180,E1 -2934.787,E2 -2934.787} C_VEL
LIN {X 0,Y 559.154,Z 265.145,A -85,B 0,C 180,E1 -2937.364,E2 -2937.364} C_VEL
LIN {X 0,Y 559.146,Z 265.148,A -85,B 0,C 180,E1 -2940.143,E2 -2940.143} C_VEL
LIN {X 0,Y 559.196,Z 265.258,A -85,B 0,C 180,E1 -2941.408,E2 -2941.408} C_VEL
LIN {X 0,Y 562.249,Z 276.142,A -85,B 0,C 180,E1 -2942.558,E2 -2942.558} C_VEL
LIN {X 0,Y 561.812,Z 301.706,A -85,B 0,C 180,E1 -2944.829,E2 -2944.829} C_VEL
LIN {X 0,Y 561.68,Z 312.356,A -85,B 0,C 180,E1 -2945.743,E2 -2945.743} C_VEL
LIN {X 0,Y 563.221,Z 321.181,A -85,B 0,C 180,E1 -2945.934,E2 -2945.934} C_VEL
LIN {X 0,Y 562.293,Z 517.938,A -85,B 0,C 180,E1 -2948.58,E2 -2948.58} C_VEL
LIN {X 0,Y 562.073,Z 534.177,A -85,B 0,C 180,E1 -2948.932,E2 -2948.932} C_VEL
LIN {X 0,Y 561.787,Z 550.94,A -85,B 0,C 180,E1 -2949.448,E2 -2949.448} C_VEL
LIN {X 0,Y 561.501,Z 565.854,A -85,B 0,C 180,E1 -2950.045,E2 -2950.045} C_VEL
LIN {X 0,Y 561.137,Z 581.034,A -85,B 0,C 180,E1 -2950.806,E2 -2950.806} C_VEL
LIN {X 0,Y 560.779,Z 594.849,A -85,B 0,C 180,E1 -2951.646,E2 -2951.646} C_VEL
LIN {X 0,Y 560.367,Z 609.043,A -85,B 0,C 180,E1 -2952.671,E2 -2952.671} C_VEL
LIN {X 0,Y 559.988,Z 622.118,A -85,B 0,C 180,E1 -2953.785,E2 -2953.785} C_VEL
LIN {X 0,Y 559.722,Z 634.654,A -85,B 0,C 180,E1 -2955.044,E2 -2955.044} C_VEL
LIN {X 0,Y 559.448,Z 645.907,A -85,B 0,C 180,E1 -2956.376,E2 -2956.376} C_VEL
LIN {X 0,Y 559.219,Z 656.441,A -85,B 0,C 180,E1 -2957.848,E2 -2957.848} C_VEL
LIN {X 0,Y 559.057,Z 665.276,A -85,B 0,C 180,E1 -2959.314,E2 -2959.314} C_VEL
LIN {X 0,Y 558.93,Z 671.856,A -85,B 0,C 180,E1 -2960.592,E2 -2960.592} C_VEL
LIN {X 0,Y 558.893,Z 679.466,A -85,B 0,C 180,E1 -2962.413,E2 -2962.413} C_VEL
LIN {X 0,Y 558.863,Z 685.248,A -85,B 0,C 180,E1 -2964.226,E2 -2964.226} C_VEL
LIN {X 0,Y 558.805,Z 688.636,A -85,B 0,C 180,E1 -2965.672,E2 -2965.672} C_VEL
LIN {X 0,Y 558.787,Z 691.09,A -85,B 0,C 180,E1 -2967.116,E2 -2967.116} C_VEL
LIN {X 0,Y 558.739,Z 692.48,A -85,B 0,C 180,E1 -2968.559,E2 -2968.559} C_VEL
LIN {X 0,Y 558.735,Z 693,A -85,B 0,C 180,E1 -2970,E2 -2970} C_VEL
LIN {X 0,Y 558.738,Z 692.479,A -85,B 0,C 180,E1 -2971.442,E2 -2971.442} C_VEL
LIN {X 0,Y 558.787,Z 691.088,A -85,B 0,C 180,E1 -2972.884,E2 -2972.884} C_VEL
LIN {X 0,Y 558.805,Z 688.635,A -85,B 0,C 180,E1 -2974.328,E2 -2974.328} C_VEL
LIN {X 0,Y 558.862,Z 685.249,A -85,B 0,C 180,E1 -2975.774,E2 -2975.774} C_VEL
LIN {X 0,Y 558.893,Z 679.467,A -85,B 0,C 180,E1 -2977.587,E2 -2977.587} C_VEL
LIN {X 0,Y 558.93,Z 671.856,A -85,B 0,C 180,E1 -2979.408,E2 -2979.408} C_VEL
LIN {X 0,Y 559.116,Z 663.28,A -85,B 0,C 180,E1 -2981.046,E2 -2981.046} C_VEL
LIN {X 0,Y 559.275,Z 653.975,A -85,B 0,C 180,E1 -2982.519,E2 -2982.519} C_VEL
LIN {X 0,Y 559.471,Z 644.421,A -85,B 0,C 180,E1 -2983.808,E2 -2983.808} C_VEL
LIN {X 0,Y 559.791,Z 633.258,A -85,B 0,C 180,E1 -2985.103,E2 -2985.103} C_VEL
LIN {X 0,Y 560.05,Z 621.139,A -85,B 0,C 180,E1 -2986.307,E2 -2986.307} C_VEL
LIN {X 0,Y 560.42,Z 607.868,A -85,B 0,C 180,E1 -2987.422,E2 -2987.422} C_VEL
LIN {X 0,Y 560.786,Z 594.845,A -85,B 0,C 180,E1 -2988.353,E2 -2988.353} C_VEL
LIN {X 0,Y 561.133,Z 581.026,A -85,B 0,C 180,E1 -2989.194,E2 -2989.194} C_VEL
LIN {X 0,Y 561.469,Z 566.936,A -85,B 0,C 180,E1 -2989.904,E2 -2989.904} C_VEL
LIN {X 0,Y 561.773,Z 550.936,A -85,B 0,C 180,E1 -2990.553,E2 -2990.553} C_VEL
LIN {X 0,Y 562.11,Z 534.176,A -85,B 0,C 180,E1 -2991.067,E2 -2991.067} C_VEL
LIN {X 0,Y 562.273,Z 517.929,A -85,B 0,C 180,E1 -2991.421,E2 -2991.421} C_VEL
LIN {X 0,Y 563.202,Z 320.984,A -85,B 0,C 180,E1 -2994.07,E2 -2994.07} C_VEL
LIN {X 0,Y 561.619,Z 311.974,A -85,B 0,C 180,E1 -2994.27,E2 -2994.27} C_VEL
LIN {X 0,Y 562.279,Z 278.273,A -85,B 0,C 180,E1 -2997.243,E2 -2997.243} C_VEL
LIN {X 0,Y 562.04,Z 274.903,A -85,B 0,C 180,E1 -2997.559,E2 -2997.559} C_VEL
LIN {X 0,Y 559.175,Z 265.146,A -85,B 0,C 180,E1 -2998.606,E2 -2998.606} C_VEL
LIN {X 0,Y 559.148,Z 265.15,A -85,B 0,C 180,E1 -3001.274,E2 -3001.274} C_VEL
LIN {X 0,Y 559.165,Z 265.143,A -85,B 0,C 180,E1 -3003.949,E2 -3003.949} C_VEL
LIN {X 0,Y 559.14,Z 265.15,A -85,B 0,C 180,E1 -3007.109,E2 -3007.109} C_VEL
LIN {X 0,Y 559.164,Z 265.142,A -85,B 0,C 180,E1 -3009.943,E2 -3009.943} C_VEL
LIN {X 0,Y 559.163,Z 265.143,A -85,B 0,C 180,E1 -3012.743,E2 -3012.743} C_VEL
LIN {X 0,Y 559.153,Z 265.143,A -85,B 0,C 180,E1 -3015.761,E2 -3015.761} C_VEL
LIN {X 0,Y 559.192,Z 265.136,A -85,B 0,C 180,E1 -3018.233,E2 -3018.233} C_VEL
LIN {X 0,Y 559.179,Z 265.144,A -85,B 0,C 180,E1 -3021.192,E2 -3021.192} C_VEL
LIN {X 0,Y 559.14,Z 265.144,A -85,B 0,C 180,E1 -3023.79,E2 -3023.79} C_VEL
LIN {X 0,Y 559.163,Z 265.142,A -85,B 0,C 180,E1 -3026.426,E2 -3026.426} C_VEL
LIN {X 0,Y 559.158,Z 265.15,A -85,B 0,C 180,E1 -3028.981,E2 -3028.981} C_VEL
LIN {X 0,Y 559.169,Z 265.135,A -85,B 0,C 180,E1 -3031.619,E2 -3031.619} C_VEL
LIN {X 0,Y 559.181,Z 265.138,A -85,B 0,C 180,E1 -3033.903,E2 -3033.903} C_VEL
LIN {X 0,Y 559.152,Z 265.147,A -85,B 0,C 180,E1 -3036.569,E2 -3036.569} C_VEL
LIN {X 0,Y 559.176,Z 265.14,A -85,B 0,C 180,E1 -3039.396,E2 -3039.396} C_VEL
LIN {X 0,Y 559.141,Z 265.142,A -85,B 0,C 180,E1 -3041.686,E2 -3041.686} C_VEL
LIN {X 0,Y 559.16,Z 265.137,A -85,B 0,C 180,E1 -3043.948,E2 -3043.948} C_VEL
LIN {X 0,Y 559.165,Z 265.143,A -85,B 0,C 180,E1 -3046.184,E2 -3046.184} C_VEL
LIN {X 0,Y 559.194,Z 265.133,A -85,B 0,C 180,E1 -3049.134,E2 -3049.134} C_VEL
LIN {X 0,Y 559.193,Z 265.139,A -85,B 0,C 180,E1 -3052.054,E2 -3052.054} C_VEL
LIN {X 0,Y 559.242,Z 265.128,A -85,B 0,C 180,E1 -3054.954,E2 -3054.954} C_VEL
LIN {X 0,Y 559.253,Z 265.129,A -85,B 0,C 180,E1 -3057.84,E2 -3057.84} C_VEL
LIN {X 0,Y 559.268,Z 265.128,A -85,B 0,C 180,E1 -3060.72,E2 -3060.72} C_VEL
LIN {X 0,Y 559.223,Z 265.134,A -85,B 0,C 180,E1 -3062.882,E2 -3062.882} C_VEL
LIN {X 0,Y 559.211,Z 265.136,A -85,B 0,C 180,E1 -3065.771,E2 -3065.771} C_VEL
LIN {X 0,Y 559.164,Z 265.143,A -85,B 0,C 180,E1 -3068.675,E2 -3068.675} C_VEL
LIN {X 0,Y 559.204,Z 265.136,A -85,B 0,C 180,E1 -3071.601,E2 -3071.601} C_VEL
LIN {X 0,Y 559.184,Z 265.141,A -85,B 0,C 180,E1 -3074.588,E2 -3074.588} C_VEL
LIN {X 0,Y 559.116,Z 265.147,A -85,B 0,C 180,E1 -3077.559,E2 -3077.559} C_VEL
LIN {X 0,Y 559.162,Z 265.14,A -85,B 0,C 180,E1 -3079.838,E2 -3079.838} C_VEL
LIN {X 0,Y 559.123,Z 265.154,A -85,B 0,C 180,E1 -3082.154,E2 -3082.154} C_VEL
LIN {X 0,Y 559.131,Z 265.144,A -85,B 0,C 180,E1 -3085.176,E2 -3085.176} C_VEL
LIN {X 0,Y 559.095,Z 265.153,A -85,B 0,C 180,E1 -3087.717,E2 -3087.717} C_VEL
LIN {X 0,Y 559.105,Z 265.15,A -85,B 0,C 180,E1 -3090.605,E2 -3090.605} C_VEL
LIN {X 0,Y 558.461,Z 265.229,A -85,B 0,C 180,E1 -3091.207,E2 -3091.207} C_VEL
LIN {X 0,Y 555.604,Z 265.59,A -85,B 0,C 180,E1 -3092.183,E2 -3092.183} C_VEL
LIN {X 0,Y 553.182,Z 265.888,A -85,B 0,C 180,E1 -3092.969,E2 -3092.969} C_VEL
LIN {X 0,Y 552.151,Z 266.018,A -85,B 0,C 180,E1 -3093.576,E2 -3093.576} C_VEL
LIN {X 0,Y 552.073,Z 266.028,A -85,B 0,C 180,E1 -3093.781,E2 -3093.781} C_VEL
LIN {X 0,Y 552.04,Z 266.03,A -85,B 0,C 180,E1 -3096.753,E2 -3096.753} C_VEL
LIN {X 0,Y 552.078,Z 266.027,A -85,B 0,C 180,E1 -3099.532,E2 -3099.532} C_VEL
LIN {X 0,Y 552.082,Z 266.026,A -85,B 0,C 180,E1 -3102.431,E2 -3102.431} C_VEL
LIN {X 0,Y 552.075,Z 266.029,A -85,B 0,C 180,E1 -3105.56,E2 -3105.56} C_VEL
LIN {X 0,Y 552.056,Z 266.029,A -85,B 0,C 180,E1 -3108.548,E2 -3108.548} C_VEL
LIN {X 0,Y 552.117,Z 266.056,A -85,B 0,C 180,E1 -3110.541,E2 -3110.541} C_VEL
LIN {X 0,Y 554.764,Z 276.338,A -85,B 0,C 180,E1 -3111.763,E2 -3111.763} C_VEL
LIN {X 0,Y 554.764,Z 283.487,A -85,B 0,C 180,E1 -3112.477,E2 -3112.477} C_VEL
LIN {X 0,Y 556.722,Z 294.157,A -85,B 0,C 180,E1 -3112.718,E2 -3112.718} C_VEL
LIN {X 0,Y 555.671,Z 488.854,A -85,B 0,C 180,E1 -3115.372,E2 -3115.372} C_VEL
LIN {X 0,Y 555.41,Z 504.875,A -85,B 0,C 180,E1 -3115.73,E2 -3115.73} C_VEL
LIN {X 0,Y 555.095,Z 521.015,A -85,B 0,C 180,E1 -3116.236,E2 -3116.236} C_VEL
LIN {X 0,Y 554.786,Z 535.987,A -85,B 0,C 180,E1 -3116.845,E2 -3116.845} C_VEL
LIN {X 0,Y 554.342,Z 551.135,A -85,B 0,C 180,E1 -3117.612,E2 -3117.612} C_VEL
LIN {X 0,Y 553.955,Z 565.774,A -85,B 0,C 180,E1 -3118.52,E2 -3118.52} C_VEL
LIN {X 0,Y 553.514,Z 579.87,A -85,B 0,C 180,E1 -3119.561,E2 -3119.561} C_VEL
LIN {X 0,Y 553.105,Z 593.034,A -85,B 0,C 180,E1 -3120.712,E2 -3120.712} C_VEL
LIN {X 0,Y 552.752,Z 605.01,A -85,B 0,C 180,E1 -3121.937,E2 -3121.937} C_VEL
LIN {X 0,Y 552.448,Z 616.918,A -85,B 0,C 180,E1 -3123.375,E2 -3123.375} C_VEL
LIN {X 0,Y 552.173,Z 627.519,A -85,B 0,C 180,E1 -3124.899,E2 -3124.899} C_VEL
LIN {X 0,Y 551.991,Z 636.526,A -85,B 0,C 180,E1 -3126.451,E2 -3126.451} C_VEL
LIN {X 0,Y 551.844,Z 643.698,A -85,B 0,C 180,E1 -3127.932,E2 -3127.932} C_VEL
LIN {X 0,Y 551.782,Z 649.939,A -85,B 0,C 180,E1 -3129.496,E2 -3129.496} C_VEL
LIN {X 0,Y 551.728,Z 654.814,A -85,B 0,C 180,E1 -3131.045,E2 -3131.045} C_VEL
LIN {X 0,Y 551.672,Z 657.706,A -85,B 0,C 180,E1 -3132.197,E2 -3132.197} C_VEL
LIN {X 0,Y 551.639,Z 660.485,A -85,B 0,C 180,E1 -3133.723,E2 -3133.723} C_VEL
LIN {X 0,Y 551.653,Z 662.437,A -85,B 0,C 180,E1 -3135.521,E2 -3135.521} C_VEL
LIN {X 0,Y 551.655,Z 662.942,A -85,B 0,C 180,E1 -3136.743,E2 -3136.743} C_VEL
LIN {X 0,Y 551.673,Z 662.651,A -85,B 0,C 180,E1 -3138.239,E2 -3138.239} C_VEL
LIN {X 0,Y 551.675,Z 661.361,A -85,B 0,C 180,E1 -3139.726,E2 -3139.726} C_VEL
LIN {X 0,Y 551.671,Z 659.075,A -85,B 0,C 180,E1 -3141.206,E2 -3141.206} C_VEL
LIN {X 0,Y 551.701,Z 655.792,A -85,B 0,C 180,E1 -3142.681,E2 -3142.681} C_VEL
LIN {X 0,Y 551.799,Z 651.427,A -85,B 0,C 180,E1 -3144.152,E2 -3144.152} C_VEL
LIN {X 0,Y 551.852,Z 646.039,A -85,B 0,C 180,E1 -3145.618,E2 -3145.618} C_VEL
LIN {X 0,Y 551.942,Z 637.578,A -85,B 0,C 180,E1 -3147.446,E2 -3147.446} C_VEL
LIN {X 0,Y 552.159,Z 628.173,A -85,B 0,C 180,E1 -3149.088,E2 -3149.088} C_VEL
LIN {X 0,Y 552.329,Z 618.163,A -85,B 0,C 180,E1 -3150.547,E2 -3150.547} C_VEL
LIN {X 0,Y 552.66,Z 607.891,A -85,B 0,C 180,E1 -3151.822,E2 -3151.822} C_VEL
LIN {X 0,Y 553.022,Z 595.963,A -85,B 0,C 180,E1 -3153.096,E2 -3153.096} C_VEL
LIN {X 0,Y 553.424,Z 582.972,A -85,B 0,C 180,E1 -3154.279,E2 -3154.279} C_VEL
LIN {X 0,Y 553.737,Z 570.017,A -85,B 0,C 180,E1 -3155.28,E2 -3155.28} C_VEL
LIN {X 0,Y 554.15,Z 556.096,A -85,B 0,C 180,E1 -3156.189,E2 -3156.189} C_VEL
LIN {X 0,Y 554.604,Z 541.046,A -85,B 0,C 180,E1 -3157.006,E2 -3157.006} C_VEL
LIN {X 0,Y 555.018,Z 525.585,A -85,B 0,C 180,E1 -3157.686,E2 -3157.686} C_VEL
LIN {X 0,Y 555.371,Z 508.798,A -85,B 0,C 180,E1 -3158.253,E2 -3158.253} C_VEL
LIN {X 0,Y 555.653,Z 492.823,A -85,B 0,C 180,E1 -3158.638,E2 -3158.638} C_VEL
LIN {X 0,Y 555.809,Z 471.374,A -85,B 0,C 180,E1 -3158.972,E2 -3158.972} C_VEL
LIN {X 0,Y 556.685,Z 292.875,A -85,B 0,C 180,E1 -3161.391,E2 -3161.391} C_VEL
LIN {X 0,Y 554.684,Z 282.872,A -85,B 0,C 180,E1 -3161.65,E2 -3161.65} C_VEL
LIN {X 0,Y 554.617,Z 275.3,A -85,B 0,C 180,E1 -3162.44,E2 -3162.44} C_VEL
LIN {X 0,Y 552.108,Z 266.027,A -85,B 0,C 180,E1 -3163.574,E2 -3163.574} C_VEL
LIN {X 0,Y 552.087,Z 266.03,A -85,B 0,C 180,E1 -3166.264,E2 -3166.264} C_VEL
LIN {X 0,Y 552.143,Z 266.017,A -85,B 0,C 180,E1 -3169.326,E2 -3169.326} C_VEL
LIN {X 0,Y 552.115,Z 266.021,A -85,B 0,C 180,E1 -3171.683,E2 -3171.683} C_VEL
LIN {X 0,Y 552.083,Z 266.031,A -85,B 0,C 180,E1 -3174.039,E2 -3174.039} C_VEL
LIN {X 0,Y 552.076,Z 266.024,A -85,B 0,C 180,E1 -3176.986,E2 -3176.986} C_VEL
LIN {X 0,Y 552.088,Z 266.03,A -85,B 0,C 180,E1 -3180.044,E2 -3180.044} C_VEL
LIN {X 0,Y 552.097,Z 266.022,A -85,B 0,C 180,E1 -3182.842,E2 -3182.842} C_VEL
LIN {X 0,Y 552.049,Z 266.031,A -85,B 0,C 180,E1 -3185.846,E2 -3185.846} C_VEL
LIN {X 0,Y 552.071,Z 266.023,A -85,B 0,C 180,E1 -3189.054,E2 -3189.054} C_VEL
LIN {X 0,Y 552.081,Z 266.025,A -85,B 0,C 180,E1 -3192.409,E2 -3192.409} C_VEL
LIN {X 0,Y 552.066,Z 266.028,A -85,B 0,C 180,E1 -3195.559,E2 -3195.559} C_VEL
LIN {X 0,Y 552.052,Z 266.028,A -85,B 0,C 180,E1 -3198.547,E2 -3198.547} C_VEL
LIN {X 0,Y 552.111,Z 266.02,A -85,B 0,C 180,E1 -3201.41,E2 -3201.41} C_VEL
LIN {X 0,Y 552.061,Z 266.02,A -85,B 0,C 180,E1 -3204.563,E2 -3204.563} C_VEL
LIN {X 0,Y 552.098,Z 266.021,A -85,B 0,C 180,E1 -3207.156,E2 -3207.156} C_VEL
LIN {X 0,Y 552.09,Z 266.025,A -85,B 0,C 180,E1 -3209.954,E2 -3209.954} C_VEL
LIN {X 0,Y 552.077,Z 266.024,A -85,B 0,C 180,E1 -3213.013,E2 -3213.013} C_VEL
LIN {X 0,Y 552.087,Z 266.025,A -85,B 0,C 180,E1 -3215.961,E2 -3215.961} C_VEL
LIN {X 0,Y 552.118,Z 266.02,A -85,B 0,C 180,E1 -3219.119,E2 -3219.119} C_VEL
LIN {X 0,Y 552.088,Z 266.027,A -85,B 0,C 180,E1 -3221.443,E2 -3221.443} C_VEL
LIN {X 0,Y 552.095,Z 266.029,A -85,B 0,C 180,E1 -3223.736,E2 -3223.736} C_VEL
LIN {X 0,Y 552.128,Z 266.019,A -85,B 0,C 180,E1 -3226.004,E2 -3226.004} C_VEL
LIN {X 0,Y 552.162,Z 266.011,A -85,B 0,C 180,E1 -3228.993,E2 -3228.993} C_VEL
LIN {X 0,Y 552.134,Z 266.019,A -85,B 0,C 180,E1 -3231.951,E2 -3231.951} C_VEL
LIN {X 0,Y 552.223,Z 266.003,A -85,B 0,C 180,E1 -3234.888,E2 -3234.888} C_VEL
LIN {X 0,Y 552.226,Z 266.008,A -85,B 0,C 180,E1 -3237.812,E2 -3237.812} C_VEL
LIN {X 0,Y 552.235,Z 266,A -85,B 0,C 180,E1 -3240.729,E2 -3240.729} C_VEL
LIN {X 0,Y 552.198,Z 266.01,A -85,B 0,C 180,E1 -3242.918,E2 -3242.918} C_VEL
LIN {X 0,Y 552.199,Z 266.007,A -85,B 0,C 180,E1 -3245.843,E2 -3245.843} C_VEL
LIN {X 0,Y 552.156,Z 266.013,A -85,B 0,C 180,E1 -3248.785,E2 -3248.785} C_VEL
LIN {X 0,Y 552.164,Z 266.014,A -85,B 0,C 180,E1 -3251.75,E2 -3251.75} C_VEL
LIN {X 0,Y 552.129,Z 266.02,A -85,B 0,C 180,E1 -3254.748,E2 -3254.748} C_VEL
LIN {X 0,Y 552.1,Z 266.022,A -85,B 0,C 180,E1 -3257.788,E2 -3257.788} C_VEL
LIN {X 0,Y 552.126,Z 266.017,A -85,B 0,C 180,E1 -3260.101,E2 -3260.101} C_VEL
LIN {X 0,Y 552.095,Z 266.021,A -85,B 0,C 180,E1 -3262.45,E2 -3262.45} C_VEL
LIN {X 0,Y 552.155,Z 266.02,A -85,B 0,C 180,E1 -3265.35,E2 -3265.35} C_VEL
LIN {X 0,Y 552.109,Z 266.019,A -85,B 0,C 180,E1 -3268.098,E2 -3268.098} C_VEL
LIN {X 0,Y 552.102,Z 266.023,A -85,B 0,C 180,E1 -3270.609,E2 -3270.609} C_VEL
LIN {X 0,Y 552.114,Z 266.026,A -85,B 0,C 180,E1 -3273.186,E2 -3273.186} C_VEL
LIN {X 0,Y 552.101,Z 266.019,A -85,B 0,C 180,E1 -3275.842,E2 -3275.842} C_VEL
LIN {X 0,Y 552.125,Z 266.025,A -85,B 0,C 180,E1 -3279.062,E2 -3279.062} C_VEL
LIN {X 0,Y 552.137,Z 266.018,A -85,B 0,C 180,E1 -3281.444,E2 -3281.444} C_VEL
LIN {X 0,Y 552.094,Z 266.025,A -85,B 0,C 180,E1 -3284.532,E2 -3284.532} C_VEL
LIN {X 0,Y 552.13,Z 266.017,A -85,B 0,C 180,E1 -3287.584,E2 -3287.584} C_VEL
LIN {X 0,Y 552.131,Z 266.022,A -85,B 0,C 180,E1 -3290.473,E2 -3290.473} C_VEL
LIN {X 0,Y 552.105,Z 266.022,A -85,B 0,C 180,E1 -3293.317,E2 -3293.317} C_VEL
LIN {X 0,Y 552.125,Z 266.019,A -85,B 0,C 180,E1 -3295.939,E2 -3295.939} C_VEL
LIN {X 0,Y 552.118,Z 266.026,A -85,B 0,C 180,E1 -3298.541,E2 -3298.541} C_VEL
LIN {X 0,Y 552.114,Z 266.043,A -85,B 0,C 180,E1 -3301.098,E2 -3301.098} C_VEL
LIN {X 0,Y 555.635,Z 278.436,A -85,B 0,C 180,E1 -3302.431,E2 -3302.431} C_VEL
LIN {X 0,Y 554.987,Z 307.084,A -85,B 0,C 180,E1 -3304.999,E2 -3304.999} C_VEL
LIN {X 0,Y 554.891,Z 311.782,A -85,B 0,C 180,E1 -3305.416,E2 -3305.416} C_VEL
LIN {X 0,Y 556.739,Z 322.254,A -85,B 0,C 180,E1 -3305.653,E2 -3305.653} C_VEL
LIN {X 0,Y 555.7,Z 517.938,A -85,B 0,C 180,E1 -3308.313,E2 -3308.313} C_VEL
LIN {X 0,Y 555.444,Z 534.176,A -85,B 0,C 180,E1 -3308.668,E2 -3308.668} C_VEL
LIN {X 0,Y 555.135,Z 550.939,A -85,B 0,C 180,E1 -3309.19,E2 -3309.19} C_VEL
LIN {X 0,Y 554.821,Z 565.409,A -85,B 0,C 180,E1 -3309.773,E2 -3309.773} C_VEL
LIN {X 0,Y 554.391,Z 581.038,A -85,B 0,C 180,E1 -3310.563,E2 -3310.563} C_VEL
LIN {X 0,Y 553.961,Z 596.272,A -85,B 0,C 180,E1 -3311.508,E2 -3311.508} C_VEL
LIN {X 0,Y 553.473,Z 610.376,A -85,B 0,C 180,E1 -3312.556,E2 -3312.556} C_VEL
LIN {X 0,Y 553.046,Z 624.067,A -85,B 0,C 180,E1 -3313.765,E2 -3313.765} C_VEL
LIN {X 0,Y 552.786,Z 634.978,A -85,B 0,C 180,E1 -3314.889,E2 -3314.889} C_VEL
LIN {X 0,Y 552.445,Z 645.906,A -85,B 0,C 180,E1 -3316.2,E2 -3316.2} C_VEL
LIN {X 0,Y 552.209,Z 656.44,A -85,B 0,C 180,E1 -3317.691,E2 -3317.691} C_VEL
LIN {X 0,Y 551.992,Z 665.276,A -85,B 0,C 180,E1 -3319.176,E2 -3319.176} C_VEL
LIN {X 0,Y 551.861,Z 671.856,A -85,B 0,C 180,E1 -3320.471,E2 -3320.471} C_VEL
LIN {X 0,Y 551.803,Z 679.466,A -85,B 0,C 180,E1 -3322.315,E2 -3322.315} C_VEL
LIN {X 0,Y 551.77,Z 685.249,A -85,B 0,C 180,E1 -3324.152,E2 -3324.152} C_VEL
LIN {X 0,Y 551.702,Z 688.636,A -85,B 0,C 180,E1 -3325.617,E2 -3325.617} C_VEL
LIN {X 0,Y 551.711,Z 691.09,A -85,B 0,C 180,E1 -3327.079,E2 -3327.079} C_VEL
LIN {X 0,Y 551.638,Z 692.479,A -85,B 0,C 180,E1 -3328.54,E2 -3328.54} C_VEL
LIN {X 0,Y 551.636,Z 693,A -85,B 0,C 180,E1 -3330,E2 -3330} C_VEL
LIN {X 0,Y 551.638,Z 692.479,A -85,B 0,C 180,E1 -3331.46,E2 -3331.46} C_VEL
LIN {X 0,Y 551.711,Z 691.089,A -85,B 0,C 180,E1 -3332.921,E2 -3332.921} C_VEL
LIN {X 0,Y 551.702,Z 688.635,A -85,B 0,C 180,E1 -3334.384,E2 -3334.384} C_VEL
LIN {X 0,Y 551.77,Z 685.25,A -85,B 0,C 180,E1 -3335.849,E2 -3335.849} C_VEL
LIN {X 0,Y 551.804,Z 679.467,A -85,B 0,C 180,E1 -3337.685,E2 -3337.685} C_VEL
LIN {X 0,Y 551.86,Z 671.856,A -85,B 0,C 180,E1 -3339.53,E2 -3339.53} C_VEL
LIN {X 0,Y 552.04,Z 664.266,A -85,B 0,C 180,E1 -3341.009,E2 -3341.009} C_VEL
LIN {X 0,Y 552.226,Z 655.209,A -85,B 0,C 180,E1 -3342.495,E2 -3342.495} C_VEL
LIN {X 0,Y 552.483,Z 644.42,A -85,B 0,C 180,E1 -3343.987,E2 -3343.987} C_VEL
LIN {X 0,Y 552.855,Z 633.447,A -85,B 0,C 180,E1 -3345.277,E2 -3345.277} C_VEL
LIN {X 0,Y 553.161,Z 621.138,A -85,B 0,C 180,E1 -3346.516,E2 -3346.516} C_VEL
LIN {X 0,Y 553.578,Z 607.635,A -85,B 0,C 180,E1 -3347.663,E2 -3347.663} C_VEL
LIN {X 0,Y 553.994,Z 593.415,A -85,B 0,C 180,E1 -3348.683,E2 -3348.683} C_VEL
LIN {X 0,Y 554.414,Z 579.269,A -85,B 0,C 180,E1 -3349.533,E2 -3349.533} C_VEL
LIN {X 0,Y 554.846,Z 564.255,A -85,B 0,C 180,E1 -3350.278,E2 -3350.278} C_VEL
LIN {X 0,Y 555.218,Z 548.337,A -85,B 0,C 180,E1 -3350.904,E2 -3350.904} C_VEL
LIN {X 0,Y 555.502,Z 532.343,A -85,B 0,C 180,E1 -3351.378,E2 -3351.378} C_VEL
LIN {X 0,Y 555.683,Z 516.423,A -85,B 0,C 180,E1 -3351.712,E2 -3351.712} C_VEL
LIN {X 0,Y 556.724,Z 322.196,A -85,B 0,C 180,E1 -3354.348,E2 -3354.348} C_VEL
LIN {X 0,Y 554.898,Z 311.66,A -85,B 0,C 180,E1 -3354.592,E2 -3354.592} C_VEL
LIN {X 0,Y 555.638,Z 278.513,A -85,B 0,C 180,E1 -3357.555,E2 -3357.555} C_VEL
LIN {X 0,Y 552.114,Z 266.028,A -85,B 0,C 180,E1 -3358.902,E2 -3358.902} C_VEL
LIN {X 0,Y 552.11,Z 266.026,A -85,B 0,C 180,E1 -3361.476,E2 -3361.476} C_VEL
LIN {X 0,Y 552.132,Z 266.018,A -85,B 0,C 180,E1 -3364.171,E2 -3364.171} C_VEL
LIN {X 0,Y 552.104,Z 266.024,A -85,B 0,C 180,E1 -3366.747,E2 -3366.747} C_VEL
LIN {X 0,Y 552.132,Z 266.022,A -85,B 0,C 180,E1 -3369.527,E2 -3369.527} C_VEL
LIN {X 0,Y 552.131,Z 266.016,A -85,B 0,C 180,E1 -3372.426,E2 -3372.426} C_VEL
LIN {X 0,Y 552.098,Z 266.023,A -85,B 0,C 180,E1 -3375.563,E2 -3375.563} C_VEL
LIN {X 0,Y 552.141,Z 266.018,A -85,B 0,C 180,E1 -3378.676,E2 -3378.676} C_VEL
LIN {X 0,Y 552.121,Z 266.02,A -85,B 0,C 180,E1 -3381.412,E2 -3381.412} C_VEL
LIN {X 0,Y 552.086,Z 266.022,A -85,B 0,C 180,E1 -3384.157,E2 -3384.157} C_VEL
LIN {X 0,Y 552.116,Z 266.023,A -85,B 0,C 180,E1 -3386.815,E2 -3386.815} C_VEL
LIN {X 0,Y 552.105,Z 266.022,A -85,B 0,C 180,E1 -3389.391,E2 -3389.391} C_VEL
LIN {X 0,Y 552.11,Z 266.013,A -85,B 0,C 180,E1 -3391.902,E2 -3391.902} C_VEL
LIN {X 0,Y 552.157,Z 266.02,A -85,B 0,C 180,E1 -3394.65,E2 -3394.65} C_VEL
LIN {X 0,Y 552.093,Z 266.017,A -85,B 0,C 180,E1 -3397.549,E2 -3397.549} C_VEL
LIN {X 0,Y 552.146,Z 266.019,A -85,B 0,C 180,E1 -3400.375,E2 -3400.375} C_VEL
LIN {X 0,Y 552.135,Z 266.016,A -85,B 0,C 180,E1 -3402.977,E2 -3402.977} C_VEL
LIN {X 0,Y 552.132,Z 266.018,A -85,B 0,C 180,E1 -3406.005,E2 -3406.005} C_VEL
LIN {X 0,Y 552.162,Z 266.01,A -85,B 0,C 180,E1 -3408.994,E2 -3408.994} C_VEL
LIN {X 0,Y 552.148,Z 266.015,A -85,B 0,C 180,E1 -3411.952,E2 -3411.952} C_VEL
LIN {X 0,Y 552.218,Z 266.003,A -85,B 0,C 180,E1 -3414.889,E2 -3414.889} C_VEL
LIN {X 0,Y 552.224,Z 266.005,A -85,B 0,C 180,E1 -3417.812,E2 -3417.812} C_VEL
LIN {X 0,Y 552.239,Z 266.003,A -85,B 0,C 180,E1 -3420.73,E2 -3420.73} C_VEL
LIN {X 0,Y 552.189,Z 266.01,A -85,B 0,C 180,E1 -3422.919,E2 -3422.919} C_VEL
LIN {X 0,Y 552.182,Z 266.013,A -85,B 0,C 180,E1 -3425.844,E2 -3425.844} C_VEL
LIN {X 0,Y 552.136,Z 266.017,A -85,B 0,C 180,E1 -3428.786,E2 -3428.786} C_VEL
LIN {X 0,Y 552.16,Z 266.015,A -85,B 0,C 180,E1 -3431.751,E2 -3431.751} C_VEL
LIN {X 0,Y 552.131,Z 266.018,A -85,B 0,C 180,E1 -3434.749,E2 -3434.749} C_VEL
LIN {X 0,Y 552.08,Z 266.026,A -85,B 0,C 180,E1 -3437.79,E2 -3437.79} C_VEL
LIN {X 0,Y 552.121,Z 266.021,A -85,B 0,C 180,E1 -3440.102,E2 -3440.102} C_VEL
LIN {X 0,Y 552.059,Z 266.029,A -85,B 0,C 180,E1 -3442.453,E2 -3442.453} C_VEL
LIN {X 0,Y 552.072,Z 266.024,A -85,B 0,C 180,E1 -3445.331,E2 -3445.331} C_VEL
LIN {X 0,Y 552.046,Z 266.032,A -85,B 0,C 180,E1 -3448.102,E2 -3448.102} C_VEL
LIN {X 0,Y 552.073,Z 266.026,A -85,B 0,C 180,E1 -3450.612,E2 -3450.612} C_VEL
LIN {X 0,Y 552.09,Z 266.022,A -85,B 0,C 180,E1 -3453.188,E2 -3453.188} C_VEL
LIN {X 0,Y 552.073,Z 266.028,A -85,B 0,C 180,E1 -3453.781,E2 -3453.781} C_VEL
LIN {X 0,Y 551.417,Z 266.115,A -85,B 0,C 180,E1 -3454.39,E2 -3454.39} C_VEL
LIN {X 0,Y 548.545,Z 266.472,A -85,B 0,C 180,E1 -3455.378,E2 -3455.378} C_VEL
LIN {X 0,Y 546.111,Z 266.775,A -85,B 0,C 180,E1 -3456.173,E2 -3456.173} C_VEL
LIN {X 0,Y 545.07,Z 266.899,A -85,B 0,C 180,E1 -3456.787,E2 -3456.787} C_VEL
LIN {X 0,Y 544.988,Z 266.909,A -85,B 0,C 180,E1 -3456.995,E2 -3456.995} C_VEL
LIN {X 0,Y 545.034,Z 266.903,A -85,B 0,C 180,E1 -3459.315,E2 -3459.315} C_VEL
LIN {X 0,Y 545.031,Z 266.908,A -85,B 0,C 180,E1 -3462.108,E2 -3462.108} C_VEL
LIN {X 0,Y 545.021,Z 266.905,A -85,B 0,C 180,E1 -3465.172,E2 -3465.172} C_VEL
LIN {X 0,Y 545.033,Z 266.909,A -85,B 0,C 180,E1 -3467.893,E2 -3467.893} C_VEL
LIN {X 0,Y 545.089,Z 267.082,A -85,B 0,C 180,E1 -3470.259,E2 -3470.259} C_VEL
LIN {X 0,Y 547.868,Z 277.219,A -85,B 0,C 180,E1 -3471.491,E2 -3471.491} C_VEL
LIN {X 0,Y 548.07,Z 282.057,A -85,B 0,C 180,E1 -3472.011,E2 -3472.011} C_VEL
LIN {X 0,Y 548.119,Z 283.711,A -85,B 0,C 180,E1 -3472.159,E2 -3472.159} C_VEL
LIN {X 0,Y 550.28,Z 294.824,A -85,B 0,C 180,E1 -3472.421,E2 -3472.421} C_VEL
LIN {X 0,Y 549.083,Z 489.37,A -85,B 0,C 180,E1 -3475.105,E2 -3475.105} C_VEL
LIN {X 0,Y 548.796,Z 506.043,A -85,B 0,C 180,E1 -3475.489,E2 -3475.489} C_VEL
LIN {X 0,Y 548.415,Z 522.111,A -85,B 0,C 180,E1 -3476.009,E2 -3476.009} C_VEL
LIN {X 0,Y 548.029,Z 538.321,A -85,B 0,C 180,E1 -3476.699,E2 -3476.699} C_VEL
LIN {X 0,Y 547.576,Z 552.919,A -85,B 0,C 180,E1 -3477.467,E2 -3477.467} C_VEL
LIN {X 0,Y 547.133,Z 566.482,A -85,B 0,C 180,E1 -3478.329,E2 -3478.329} C_VEL
LIN {X 0,Y 546.67,Z 579.677,A -85,B 0,C 180,E1 -3479.32,E2 -3479.32} C_VEL
LIN {X 0,Y 546.193,Z 593.205,A -85,B 0,C 180,E1 -3480.516,E2 -3480.516} C_VEL
LIN {X 0,Y 545.801,Z 605.154,A -85,B 0,C 180,E1 -3481.757,E2 -3481.757} C_VEL
LIN {X 0,Y 545.447,Z 616.903,A -85,B 0,C 180,E1 -3483.194,E2 -3483.194} C_VEL
LIN {X 0,Y 545.188,Z 626.896,A -85,B 0,C 180,E1 -3484.645,E2 -3484.645} C_VEL
LIN {X 0,Y 544.992,Z 634.875,A -85,B 0,C 180,E1 -3486.005,E2 -3486.005} C_VEL
LIN {X 0,Y 544.804,Z 642.915,A -85,B 0,C 180,E1 -3487.632,E2 -3487.632} C_VEL
LIN {X 0,Y 544.705,Z 649.315,A -85,B 0,C 180,E1 -3489.218,E2 -3489.218} C_VEL
LIN {X 0,Y 544.64,Z 654.306,A -85,B 0,C 180,E1 -3490.789,E2 -3490.789} C_VEL
LIN {X 0,Y 544.57,Z 657.288,A -85,B 0,C 180,E1 -3491.957,E2 -3491.957} C_VEL
LIN {X 0,Y 544.562,Z 660.22,A -85,B 0,C 180,E1 -3493.505,E2 -3493.505} C_VEL
LIN {X 0,Y 544.51,Z 662.121,A -85,B 0,C 180,E1 -3495.04,E2 -3495.04} C_VEL
LIN {X 0,Y 544.553,Z 662.905,A -85,B 0,C 180,E1 -3496.567,E2 -3496.567} C_VEL
LIN {X 0,Y 544.566,Z 662.76,A -85,B 0,C 180,E1 -3498.083,E2 -3498.083} C_VEL
LIN {X 0,Y 544.579,Z 661.544,A -85,B 0,C 180,E1 -3499.591,E2 -3499.591} C_VEL
LIN {X 0,Y 544.565,Z 659.405,A -85,B 0,C 180,E1 -3501.091,E2 -3501.091} C_VEL
LIN {X 0,Y 544.611,Z 656.2,A -85,B 0,C 180,E1 -3502.585,E2 -3502.585} C_VEL
LIN {X 0,Y 544.71,Z 651.991,A -85,B 0,C 180,E1 -3504.075,E2 -3504.075} C_VEL
LIN {X 0,Y 544.781,Z 646.686,A -85,B 0,C 180,E1 -3505.561,E2 -3505.561} C_VEL
LIN {X 0,Y 544.803,Z 640.203,A -85,B 0,C 180,E1 -3507.042,E2 -3507.042} C_VEL
LIN {X 0,Y 545.029,Z 632.475,A -85,B 0,C 180,E1 -3508.522,E2 -3508.522} C_VEL
LIN {X 0,Y 545.235,Z 623.272,A -85,B 0,C 180,E1 -3510,E2 -3510} C_VEL
LIN {X 0,Y 545.457,Z 613.823,A -85,B 0,C 180,E1 -3511.292,E2 -3511.292} C_VEL
LIN {X 0,Y 545.886,Z 602.883,A -85,B 0,C 180,E1 -3512.583,E2 -3512.583} C_VEL
LIN {X 0,Y 546.242,Z 592.027,A -85,B 0,C 180,E1 -3513.688,E2 -3513.688} C_VEL
LIN {X 0,Y 546.632,Z 579.407,A -85,B 0,C 180,E1 -3514.794,E2 -3514.794} C_VEL
LIN {X 0,Y 547.063,Z 565.86,A -85,B 0,C 180,E1 -3515.806,E2 -3515.806} C_VEL
LIN {X 0,Y 547.563,Z 551.193,A -85,B 0,C 180,E1 -3516.726,E2 -3516.726} C_VEL
LIN {X 0,Y 548.083,Z 535.015,A -85,B 0,C 180,E1 -3517.552,E2 -3517.552} C_VEL
LIN {X 0,Y 548.506,Z 518.987,A -85,B 0,C 180,E1 -3518.195,E2 -3518.195} C_VEL
LIN {X 0,Y 548.845,Z 503.141,A -85,B 0,C 180,E1 -3518.677,E2 -3518.677} C_VEL
LIN {X 0,Y 549.094,Z 485.723,A -85,B 0,C 180,E1 -3519.044,E2 -3519.044} C_VEL
LIN {X 0,Y 550.242,Z 294.434,A -85,B 0,C 180,E1 -3521.675,E2 -3521.675} C_VEL
LIN {X 0,Y 548.014,Z 283.274,A -85,B 0,C 180,E1 -3521.949,E2 -3521.949} C_VEL
LIN {X 0,Y 547.871,Z 277.185,A -85,B 0,C 180,E1 -3522.596,E2 -3522.596} C_VEL
LIN {X 0,Y 545.077,Z 266.905,A -85,B 0,C 180,E1 -3523.847,E2 -3523.847} C_VEL
LIN {X 0,Y 545.04,Z 266.908,A -85,B 0,C 180,E1 -3526.48,E2 -3526.48} C_VEL
LIN {X 0,Y 545.108,Z 266.895,A -85,B 0,C 180,E1 -3529.586,E2 -3529.586} C_VEL
LIN {X 0,Y 545.031,Z 266.905,A -85,B 0,C 180,E1 -3532.758,E2 -3532.758} C_VEL
LIN {X 0,Y 545.031,Z 266.902,A -85,B 0,C 180,E1 -3535.493,E2 -3535.493} C_VEL
LIN {X 0,Y 545.034,Z 266.906,A -85,B 0,C 180,E1 -3538.496,E2 -3538.496} C_VEL
LIN {X 0,Y 545.042,Z 266.901,A -85,B 0,C 180,E1 -3541.049,E2 -3541.049} C_VEL
LIN {X 0,Y 545.036,Z 266.904,A -85,B 0,C 180,E1 -3543.674,E2 -3543.674} C_VEL
LIN {X 0,Y 544.989,Z 266.911,A -85,B 0,C 180,E1 -3546.384,E2 -3546.384} C_VEL
LIN {X 0,Y 545.021,Z 266.902,A -85,B 0,C 180,E1 -3549.312,E2 -3549.312} C_VEL
LIN {X 0,Y 545.029,Z 266.907,A -85,B 0,C 180,E1 -3552.108,E2 -3552.108} C_VEL
LIN {X 0,Y 545.014,Z 266.903,A -85,B 0,C 180,E1 -3555.172,E2 -3555.172} C_VEL
LIN {X 0,Y 545.021,Z 266.905,A -85,B 0,C 180,E1 -3558.409,E2 -3558.409} C_VEL
LIN {X 0,Y 545.065,Z 266.894,A -85,B 0,C 180,E1 -3560.816,E2 -3560.816} C_VEL
LIN {X 0,Y 545.001,Z 266.899,A -85,B 0,C 180,E1 -3563.616,E2 -3563.616} C_VEL
LIN {X 0,Y 545.052,Z 266.9,A -85,B 0,C 180,E1 -3566.327,E2 -3566.327} C_VEL
LIN {X 0,Y 545.055,Z 266.898,A -85,B 0,C 180,E1 -3568.951,E2 -3568.951} C_VEL
LIN {X 0,Y 545.034,Z 266.902,A -85,B 0,C 180,E1 -3571.503,E2 -3571.503} C_VEL
LIN {X 0,Y 545.034,Z 266.9,A -85,B 0,C 180,E1 -3574.505,E2 -3574.505} C_VEL
LIN {X 0,Y 545.035,Z 266.9,A -85,B 0,C 180,E1 -3577.242,E2 -3577.242} C_VEL
LIN {X 0,Y 545.118,Z 266.89,A -85,B 0,C 180,E1 -3580.414,E2 -3580.414} C_VEL
LIN {X 0,Y 545.047,Z 266.904,A -85,B 0,C 180,E1 -3583.52,E2 -3583.52} C_VEL
LIN {X 0,Y 545.083,Z 266.899,A -85,B 0,C 180,E1 -3585.819,E2 -3585.819} C_VEL
LIN {X 0,Y 545.118,Z 266.887,A -85,B 0,C 180,E1 -3588.849,E2 -3588.849} C_VEL
LIN {X 0,Y 545.086,Z 266.898,A -85,B 0,C 180,E1 -3591.846,E2 -3591.846} C_VEL
LIN {X 0,Y 545.164,Z 266.882,A -85,B 0,C 180,E1 -3594.08,E2 -3594.08} C_VEL
LIN {X 0,Y 545.161,Z 266.888,A -85,B 0,C 180,E1 -3597.044,E2 -3597.044} C_VEL
LIN {X 0,Y 545.203,Z 266.877,A -85,B 0,C 180,E1 -3600,E2 -3600} C_VEL
LIN {X 0,Y 545.166,Z 266.887,A -85,B 0,C 180,E1 -3602.955,E2 -3602.955} C_VEL
LIN {X 0,Y 545.169,Z 266.881,A -85,B 0,C 180,E1 -3605.919,E2 -3605.919} C_VEL
LIN {X 0,Y 545.116,Z 266.891,A -85,B 0,C 180,E1 -3608.9,E2 -3608.9} C_VEL
LIN {X 0,Y 545.136,Z 266.888,A -85,B 0,C 180,E1 -3611.904,E2 -3611.904} C_VEL
LIN {X 0,Y 545.082,Z 266.9,A -85,B 0,C 180,E1 -3614.943,E2 -3614.943} C_VEL
LIN {X 0,Y 545.071,Z 266.896,A -85,B 0,C 180,E1 -3618.026,E2 -3618.026} C_VEL
LIN {X 0,Y 545.092,Z 266.894,A -85,B 0,C 180,E1 -3620.372,E2 -3620.372} C_VEL
LIN {X 0,Y 545.092,Z 266.897,A -85,B 0,C 180,E1 -3623.558,E2 -3623.558} C_VEL
LIN {X 0,Y 545.079,Z 266.896,A -85,B 0,C 180,E1 -3626,E2 -3626} C_VEL
LIN {X 0,Y 545.089,Z 266.898,A -85,B 0,C 180,E1 -3628.748,E2 -3628.748} C_VEL
LIN {X 0,Y 545.057,Z 266.9,A -85,B 0,C 180,E1 -3631.679,E2 -3631.679} C_VEL
LIN {X 0,Y 545.076,Z 266.899,A -85,B 0,C 180,E1 -3634.563,E2 -3634.563} C_VEL
LIN {X 0,Y 545.038,Z 266.904,A -85,B 0,C 180,E1 -3637.303,E2 -3637.303} C_VEL
LIN {X 0,Y 545.074,Z 266.896,A -85,B 0,C 180,E1 -3640.141,E2 -3640.141} C_VEL
LIN {X 0,Y 545.077,Z 266.901,A -85,B 0,C 180,E1 -3643.106,E2 -3643.106} C_VEL
LIN {X 0,Y 545.064,Z 266.899,A -85,B 0,C 180,E1 -3646.224,E2 -3646.224} C_VEL
LIN {X 0,Y 545.096,Z 266.902,A -85,B 0,C 180,E1 -3648.887,E2 -3648.887} C_VEL
LIN {X 0,Y 545.052,Z 266.899,A -85,B 0,C 180,E1 -3651.763,E2 -3651.763} C_VEL
LIN {X 0,Y 545.035,Z 266.906,A -85,B 0,C 180,E1 -3654.532,E2 -3654.532} C_VEL
LIN {X 0,Y 545.067,Z 266.902,A -85,B 0,C 180,E1 -3657.211,E2 -3657.211} C_VEL
LIN {X 0,Y 545.062,Z 266.901,A -85,B 0,C 180,E1 -3659.81,E2 -3659.81} C_VEL
LIN {X 0,Y 545.073,Z 267.001,A -85,B 0,C 180,E1 -3660.798,E2 -3660.798} C_VEL
LIN {X 0,Y 548.838,Z 279.625,A -85,B 0,C 180,E1 -3662.189,E2 -3662.189} C_VEL
LIN {X 0,Y 548.792,Z 289.076,A -85,B 0,C 180,E1 -3663.062,E2 -3663.062} C_VEL
LIN {X 0,Y 548.242,Z 311.943,A -85,B 0,C 180,E1 -3665.108,E2 -3665.108} C_VEL
LIN {X 0,Y 550.268,Z 322.846,A -85,B 0,C 180,E1 -3665.359,E2 -3665.359} C_VEL
LIN {X 0,Y 549.091,Z 519.302,A -85,B 0,C 180,E1 -3668.063,E2 -3668.063} C_VEL
LIN {X 0,Y 548.827,Z 535.014,A -85,B 0,C 180,E1 -3668.423,E2 -3668.423} C_VEL
LIN {X 0,Y 548.48,Z 550.914,A -85,B 0,C 180,E1 -3668.926,E2 -3668.926} C_VEL
LIN {X 0,Y 548.112,Z 566.18,A -85,B 0,C 180,E1 -3669.553,E2 -3669.553} C_VEL
LIN {X 0,Y 547.662,Z 581.041,A -85,B 0,C 180,E1 -3670.314,E2 -3670.314} C_VEL
LIN {X 0,Y 547.153,Z 596.269,A -85,B 0,C 180,E1 -3671.27,E2 -3671.27} C_VEL
LIN {X 0,Y 546.63,Z 610.208,A -85,B 0,C 180,E1 -3672.317,E2 -3672.317} C_VEL
LIN {X 0,Y 546.157,Z 624.065,A -85,B 0,C 180,E1 -3673.555,E2 -3673.555} C_VEL
LIN {X 0,Y 545.837,Z 635.332,A -85,B 0,C 180,E1 -3674.734,E2 -3674.734} C_VEL
LIN {X 0,Y 545.467,Z 645.905,A -85,B 0,C 180,E1 -3676.02,E2 -3676.02} C_VEL
LIN {X 0,Y 545.182,Z 656.439,A -85,B 0,C 180,E1 -3677.53,E2 -3677.53} C_VEL
LIN {X 0,Y 544.957,Z 665.275,A -85,B 0,C 180,E1 -3679.034,E2 -3679.034} C_VEL
LIN {X 0,Y 544.795,Z 671.856,A -85,B 0,C 180,E1 -3680.346,E2 -3680.346} C_VEL
LIN {X 0,Y 544.739,Z 679.466,A -85,B 0,C 180,E1 -3682.214,E2 -3682.214} C_VEL
LIN {X 0,Y 544.686,Z 685.249,A -85,B 0,C 180,E1 -3684.075,E2 -3684.075} C_VEL
LIN {X 0,Y 544.6,Z 688.635,A -85,B 0,C 180,E1 -3685.559,E2 -3685.559} C_VEL
LIN {X 0,Y 544.638,Z 691.09,A -85,B 0,C 180,E1 -3687.041,E2 -3687.041} C_VEL
LIN {X 0,Y 544.539,Z 692.479,A -85,B 0,C 180,E1 -3688.521,E2 -3688.521} C_VEL
LIN {X 0,Y 544.536,Z 693,A -85,B 0,C 180,E1 -3690,E2 -3690} C_VEL
LIN {X 0,Y 544.539,Z 692.478,A -85,B 0,C 180,E1 -3691.479,E2 -3691.479} C_VEL
LIN {X 0,Y 544.638,Z 691.089,A -85,B 0,C 180,E1 -3692.959,E2 -3692.959} C_VEL
LIN {X 0,Y 544.6,Z 688.634,A -85,B 0,C 180,E1 -3694.441,E2 -3694.441} C_VEL
LIN {X 0,Y 544.686,Z 685.251,A -85,B 0,C 180,E1 -3695.925,E2 -3695.925} C_VEL
LIN {X 0,Y 544.739,Z 679.467,A -85,B 0,C 180,E1 -3697.786,E2 -3697.786} C_VEL
LIN {X 0,Y 544.795,Z 671.855,A -85,B 0,C 180,E1 -3699.654,E2 -3699.654} C_VEL
LIN {X 0,Y 545.017,Z 664.267,A -85,B 0,C 180,E1 -3701.153,E2 -3701.153} C_VEL
LIN {X 0,Y 545.228,Z 655.208,A -85,B 0,C 180,E1 -3702.658,E2 -3702.658} C_VEL
LIN {X 0,Y 545.53,Z 644.42,A -85,B 0,C 180,E1 -3704.169,E2 -3704.169} C_VEL
LIN {X 0,Y 545.926,Z 633.284,A -85,B 0,C 180,E1 -3705.493,E2 -3705.493} C_VEL
LIN {X 0,Y 546.263,Z 621.137,A -85,B 0,C 180,E1 -3706.73,E2 -3706.73} C_VEL
LIN {X 0,Y 546.72,Z 608.351,A -85,B 0,C 180,E1 -3707.833,E2 -3707.833} C_VEL
LIN {X 0,Y 547.169,Z 594.838,A -85,B 0,C 180,E1 -3708.827,E2 -3708.827} C_VEL
LIN {X 0,Y 547.649,Z 581.031,A -85,B 0,C 180,E1 -3709.686,E2 -3709.686} C_VEL
LIN {X 0,Y 548.126,Z 565.128,A -85,B 0,C 180,E1 -3710.498,E2 -3710.498} C_VEL
LIN {X 0,Y 548.53,Z 549.606,A -85,B 0,C 180,E1 -3711.122,E2 -3711.122} C_VEL
LIN {X 0,Y 548.874,Z 534.09,A -85,B 0,C 180,E1 -3711.6,E2 -3711.6} C_VEL
LIN {X 0,Y 549.073,Z 517.784,A -85,B 0,C 180,E1 -3711.962,E2 -3711.962} C_VEL
LIN {X 0,Y 550.245,Z 323.211,A -85,B 0,C 180,E1 -3714.637,E2 -3714.637} C_VEL
LIN {X 0,Y 548.186,Z 311.554,A -85,B 0,C 180,E1 -3714.903,E2 -3714.903} C_VEL
LIN {X 0,Y 548.987,Z 281.318,A -85,B 0,C 180,E1 -3717.638,E2 -3717.638} C_VEL
LIN {X 0,Y 548.331,Z 277.89,A -85,B 0,C 180,E1 -3717.991,E2 -3717.991} C_VEL
LIN {X 0,Y 545.083,Z 266.905,A -85,B 0,C 180,E1 -3719.221,E2 -3719.221} C_VEL
LIN {X 0,Y 545.054,Z 266.902,A -85,B 0,C 180,E1 -3721.915,E2 -3721.915} C_VEL
LIN {X 0,Y 545.061,Z 266.901,A -85,B 0,C 180,E1 -3724.565,E2 -3724.565} C_VEL
LIN {X 0,Y 545.037,Z 266.908,A -85,B 0,C 180,E1 -3727.304,E2 -3727.304} C_VEL
LIN {X 0,Y 545.071,Z 266.897,A -85,B 0,C 180,E1 -3730.142,E2 -3730.142} C_VEL
LIN {X 0,Y 545.087,Z 266.902,A -85,B 0,C 180,E1 -3733.106,E2 -3733.106} C_VEL
LIN {X 0,Y 545.067,Z 266.897,A -85,B 0,C 180,E1 -3736.225,E2 -3736.225} C_VEL
LIN {X 0,Y 545.098,Z 266.896,A -85,B 0,C 180,E1 -3738.887,E2 -3738.887} C_VEL
LIN {X 0,Y 545.054,Z 266.897,A -85,B 0,C 180,E1 -3741.763,E2 -3741.763} C_VEL
LIN {X 0,Y 545.037,Z 266.904,A -85,B 0,C 180,E1 -3744.532,E2 -3744.532} C_VEL
LIN {X 0,Y 545.069,Z 266.899,A -85,B 0,C 180,E1 -3747.212,E2 -3747.212} C_VEL
LIN {X 0,Y 545.065,Z 266.897,A -85,B 0,C 180,E1 -3749.811,E2 -3749.811} C_VEL
LIN {X 0,Y 545.082,Z 266.891,A -85,B 0,C 180,E1 -3752.344,E2 -3752.344} C_VEL
LIN {X 0,Y 545.119,Z 266.899,A -85,B 0,C 180,E1 -3754.821,E2 -3754.821} C_VEL
LIN {X 0,Y 545.041,Z 266.897,A -85,B 0,C 180,E1 -3757.243,E2 -3757.243} C_VEL
LIN {X 0,Y 545.118,Z 266.895,A -85,B 0,C 180,E1 -3760.415,E2 -3760.415} C_VEL
LIN {X 0,Y 545.063,Z 266.892,A -85,B 0,C 180,E1 -3763.521,E2 -3763.521} C_VEL
LIN {X 0,Y 545.092,Z 266.894,A -85,B 0,C 180,E1 -3765.82,E2 -3765.82} C_VEL
LIN {X 0,Y 545.118,Z 266.888,A -85,B 0,C 180,E1 -3768.85,E2 -3768.85} C_VEL
LIN {X 0,Y 545.097,Z 266.893,A -85,B 0,C 180,E1 -3771.847,E2 -3771.847} C_VEL
LIN {X 0,Y 545.195,Z 266.878,A -85,B 0,C 180,E1 -3774.823,E2 -3774.823} C_VEL
LIN {X 0,Y 545.195,Z 266.88,A -85,B 0,C 180,E1 -3777.784,E2 -3777.784} C_VEL
LIN {X 0,Y 545.209,Z 266.878,A -85,B 0,C 180,E1 -3780.739,E2 -3780.739} C_VEL
LIN {X 0,Y 545.156,Z 266.885,A -85,B 0,C 180,E1 -3782.956,E2 -3782.956} C_VEL
LIN {X 0,Y 545.132,Z 266.892,A -85,B 0,C 180,E1 -3785.92,E2 -3785.92} C_VEL
LIN {X 0,Y 545.096,Z 266.892,A -85,B 0,C 180,E1 -3788.901,E2 -3788.901} C_VEL
LIN {X 0,Y 545.103,Z 266.896,A -85,B 0,C 180,E1 -3791.905,E2 -3791.905} C_VEL
LIN {X 0,Y 545.082,Z 266.894,A -85,B 0,C 180,E1 -3794.944,E2 -3794.944} C_VEL
LIN {X 0,Y 545.05,Z 266.905,A -85,B 0,C 180,E1 -3798.027,E2 -3798.027} C_VEL
LIN {X 0,Y 545.086,Z 266.901,A -85,B 0,C 180,E1 -3800.373,E2 -3800.373} C_VEL
LIN {X 0,Y 545.074,Z 266.895,A -85,B 0,C 180,E1 -3803.56,E2 -3803.56} C_VEL
LIN {X 0,Y 545.039,Z 266.9,A -85,B 0,C 180,E1 -3806.828,E2 -3806.828} C_VEL
LIN {X 0,Y 545.016,Z 266.903,A -85,B 0,C 180,E1 -3809.342,E2 -3809.342} C_VEL
LIN {X 0,Y 545.041,Z 266.905,A -85,B 0,C 180,E1 -3811.916,E2 -3811.916} C_VEL
LIN {X 0,Y 545.041,Z 266.901,A -85,B 0,C 180,E1 -3814.567,E2 -3814.567} C_VEL
LIN {X 0,Y 544.988,Z 266.909,A -85,B 0,C 180,E1 -3816.995,E2 -3816.995} C_VEL
LIN {X 0,Y 544.329,Z 266.996,A -85,B 0,C 180,E1 -3817.612,E2 -3817.612} C_VEL
LIN {X 0,Y 541.48,Z 267.35,A -85,B 0,C 180,E1 -3818.613,E2 -3818.613} C_VEL
LIN {X 0,Y 539.067,Z 267.651,A -85,B 0,C 180,E1 -3819.419,E2 -3819.419} C_VEL
LIN {X 0,Y 538.03,Z 267.781,A -85,B 0,C 180,E1 -3820.042,E2 -3820.042} C_VEL
LIN {X 0,Y 537.945,Z 267.786,A -85,B 0,C 180,E1 -3820.253,E2 -3820.253} C_VEL
LIN {X 0,Y 537.957,Z 267.784,A -85,B 0,C 180,E1 -3822.979,E2 -3822.979} C_VEL
LIN {X 0,Y 538.002,Z 267.783,A -85,B 0,C 180,E1 -3825.929,E2 -3825.929} C_VEL
LIN {X 0,Y 537.983,Z 267.785,A -85,B 0,C 180,E1 -3828.222,E2 -3828.222} C_VEL
LIN {X 0,Y 538.024,Z 267.856,A -85,B 0,C 180,E1 -3829.94,E2 -3829.94} C_VEL
LIN {X 0,Y 541.321,Z 280.167,A -85,B 0,C 180,E1 -3831.451,E2 -3831.451} C_VEL
LIN {X 0,Y 541.422,Z 283.751,A -85,B 0,C 180,E1 -3831.827,E2 -3831.827} C_VEL
LIN {X 0,Y 543.852,Z 295.751,A -85,B 0,C 180,E1 -3832.12,E2 -3832.12} C_VEL
LIN {X 0,Y 542.505,Z 489.89,A -85,B 0,C 180,E1 -3834.832,E2 -3834.832} C_VEL
LIN {X 0,Y 542.194,Z 506.675,A -85,B 0,C 180,E1 -3835.226,E2 -3835.226} C_VEL
LIN {X 0,Y 541.769,Z 522.804,A -85,B 0,C 180,E1 -3835.759,E2 -3835.759} C_VEL
LIN {X 0,Y 541.326,Z 539.191,A -85,B 0,C 180,E1 -3836.47,E2 -3836.47} C_VEL
LIN {X 0,Y 540.821,Z 553.743,A -85,B 0,C 180,E1 -3837.254,E2 -3837.254} C_VEL
LIN {X 0,Y 540.297,Z 568.394,A -85,B 0,C 180,E1 -3838.21,E2 -3838.21} C_VEL
LIN {X 0,Y 539.754,Z 582.837,A -85,B 0,C 180,E1 -3839.347,E2 -3839.347} C_VEL
LIN {X 0,Y 539.176,Z 596.565,A -85,B 0,C 180,E1 -3840.631,E2 -3840.631} C_VEL
LIN {X 0,Y 538.737,Z 608.833,A -85,B 0,C 180,E1 -3841.989,E2 -3841.989} C_VEL
LIN {X 0,Y 538.369,Z 619.958,A -85,B 0,C 180,E1 -3843.442,E2 -3843.442} C_VEL
LIN {X 0,Y 538.09,Z 629.346,A -85,B 0,C 180,E1 -3844.882,E2 -3844.882} C_VEL
LIN {X 0,Y 537.906,Z 636.406,A -85,B 0,C 180,E1 -3846.148,E2 -3846.148} C_VEL
LIN {X 0,Y 537.724,Z 643.847,A -85,B 0,C 180,E1 -3847.726,E2 -3847.726} C_VEL
LIN {X 0,Y 537.625,Z 650.056,A -85,B 0,C 180,E1 -3849.332,E2 -3849.332} C_VEL
LIN {X 0,Y 537.551,Z 654.916,A -85,B 0,C 180,E1 -3850.922,E2 -3850.922} C_VEL
LIN {X 0,Y 537.478,Z 658.853,A -85,B 0,C 180,E1 -3852.659,E2 -3852.659} C_VEL
LIN {X 0,Y 537.432,Z 661.107,A -85,B 0,C 180,E1 -3854.061,E2 -3854.061} C_VEL
LIN {X 0,Y 537.487,Z 662.522,A -85,B 0,C 180,E1 -3855.615,E2 -3855.615} C_VEL
LIN {X 0,Y 537.473,Z 662.983,A -85,B 0,C 180,E1 -3857.156,E2 -3857.156} C_VEL
LIN {X 0,Y 537.543,Z 662.385,A -85,B 0,C 180,E1 -3858.69,E2 -3858.69} C_VEL
LIN {X 0,Y 537.48,Z 660.845,A -85,B 0,C 180,E1 -3860.213,E2 -3860.213} C_VEL
LIN {X 0,Y 537.508,Z 658.275,A -85,B 0,C 180,E1 -3861.731,E2 -3861.731} C_VEL
LIN {X 0,Y 537.609,Z 654.027,A -85,B 0,C 180,E1 -3863.481,E2 -3863.481} C_VEL
LIN {X 0,Y 537.611,Z 648.751,A -85,B 0,C 180,E1 -3865.125,E2 -3865.125} C_VEL
LIN {X 0,Y 537.73,Z 642.722,A -85,B 0,C 180,E1 -3866.628,E2 -3866.628} C_VEL
LIN {X 0,Y 537.921,Z 635.422,A -85,B 0,C 180,E1 -3868.128,E2 -3868.128} C_VEL
LIN {X 0,Y 538.132,Z 626.791,A -85,B 0,C 180,E1 -3869.626,E2 -3869.626} C_VEL
LIN {X 0,Y 538.402,Z 616.599,A -85,B 0,C 180,E1 -3871.122,E2 -3871.122} C_VEL
LIN {X 0,Y 538.851,Z 606.043,A -85,B 0,C 180,E1 -3872.429,E2 -3872.429} C_VEL
LIN {X 0,Y 539.278,Z 593.762,A -85,B 0,C 180,E1 -3873.736,E2 -3873.736} C_VEL
LIN {X 0,Y 539.77,Z 580.383,A -85,B 0,C 180,E1 -3874.948,E2 -3874.948} C_VEL
LIN {X 0,Y 540.262,Z 567.09,A -85,B 0,C 180,E1 -3875.973,E2 -3875.973} C_VEL
LIN {X 0,Y 540.817,Z 552.661,A -85,B 0,C 180,E1 -3876.904,E2 -3876.904} C_VEL
LIN {X 0,Y 541.296,Z 538.65,A -85,B 0,C 180,E1 -3877.648,E2 -3877.648} C_VEL
LIN {X 0,Y 541.79,Z 522.418,A -85,B 0,C 180,E1 -3878.344,E2 -3878.344} C_VEL
LIN {X 0,Y 542.204,Z 506.119,A -85,B 0,C 180,E1 -3878.878,E2 -3878.878} C_VEL
LIN {X 0,Y 542.524,Z 489.854,A -85,B 0,C 180,E1 -3879.257,E2 -3879.257} C_VEL
LIN {X 0,Y 543.827,Z 295.36,A -85,B 0,C 180,E1 -3881.975,E2 -3881.975} C_VEL
LIN {X 0,Y 541.362,Z 283.307,A -85,B 0,C 180,E1 -3882.295,E2 -3882.295} C_VEL
LIN {X 0,Y 541.139,Z 279.096,A -85,B 0,C 180,E1 -3882.755,E2 -3882.755} C_VEL
LIN {X 0,Y 538.064,Z 267.78,A -85,B 0,C 180,E1 -3884.176,E2 -3884.176} C_VEL
LIN {X 0,Y 538.017,Z 267.777,A -85,B 0,C 180,E1 -3887.524,E2 -3887.524} C_VEL
LIN {X 0,Y 538.03,Z 267.778,A -85,B 0,C 180,E1 -3890.652,E2 -3890.652} C_VEL
LIN {X 0,Y 538.011,Z 267.778,A -85,B 0,C 180,E1 -3893.072,E2 -3893.072} C_VEL
LIN {X 0,Y 537.99,Z 267.781,A -85,B 0,C 180,E1 -3895.659,E2 -3895.659} C_VEL
LIN {X 0,Y 537.972,Z 267.789,A -85,B 0,C 180,E1 -3898.054,E2 -3898.054} C_VEL
LIN {X 0,Y 537.998,Z 267.781,A -85,B 0,C 180,E1 -3900.628,E2 -3900.628} C_VEL
LIN {X 0,Y 538.001,Z 267.778,A -85,B 0,C 180,E1 -3903.275,E2 -3903.275} C_VEL
LIN {X 0,Y 537.944,Z 267.791,A -85,B 0,C 180,E1 -3906.008,E2 -3906.008} C_VEL
LIN {X 0,Y 537.972,Z 267.78,A -85,B 0,C 180,E1 -3908.834,E2 -3908.834} C_VEL
LIN {X 0,Y 537.975,Z 267.786,A -85,B 0,C 180,E1 -3911.871,E2 -3911.871} C_VEL
LIN {X 0,Y 537.987,Z 267.778,A -85,B 0,C 180,E1 -3914.864,E2 -3914.864} C_VEL
LIN {X 0,Y 537.961,Z 267.78,A -85,B 0,C 180,E1 -3917.208,E2 -3917.208} C_VEL
LIN {X 0,Y 537.996,Z 267.777,A -85,B 0,C 180,E1 -3920.42,E2 -3920.42} C_VEL
LIN {X 0,Y 537.954,Z 267.772,A -85,B 0,C 180,E1 -3923.061,E2 -3923.061} C_VEL
LIN {X 0,Y 538,Z 267.78,A -85,B 0,C 180,E1 -3925.825,E2 -3925.825} C_VEL
LIN {X 0,Y 537.996,Z 267.778,A -85,B 0,C 180,E1 -3928.497,E2 -3928.497} C_VEL
LIN {X 0,Y 537.985,Z 267.776,A -85,B 0,C 180,E1 -3931.095,E2 -3931.095} C_VEL
LIN {X 0,Y 537.982,Z 267.787,A -85,B 0,C 180,E1 -3933.63,E2 -3933.63} C_VEL
LIN {X 0,Y 538.008,Z 267.776,A -85,B 0,C 180,E1 -3936.122,E2 -3936.122} C_VEL
LIN {X 0,Y 538.038,Z 267.777,A -85,B 0,C 180,E1 -3939.348,E2 -3939.348} C_VEL
LIN {X 0,Y 538.038,Z 267.769,A -85,B 0,C 180,E1 -3942.467,E2 -3942.467} C_VEL
LIN {X 0,Y 538.053,Z 267.778,A -85,B 0,C 180,E1 -3945.63,E2 -3945.63} C_VEL
LIN {X 0,Y 538.078,Z 267.763,A -85,B 0,C 180,E1 -3948.701,E2 -3948.701} C_VEL
LIN {X 0,Y 538.053,Z 267.775,A -85,B 0,C 180,E1 -3951.739,E2 -3951.739} C_VEL
LIN {X 0,Y 538.119,Z 267.76,A -85,B 0,C 180,E1 -3954.002,E2 -3954.002} C_VEL
LIN {X 0,Y 538.127,Z 267.764,A -85,B 0,C 180,E1 -3957.005,E2 -3957.005} C_VEL
LIN {X 0,Y 538.174,Z 267.752,A -85,B 0,C 180,E1 -3960,E2 -3960} C_VEL
LIN {X 0,Y 538.133,Z 267.763,A -85,B 0,C 180,E1 -3962.994,E2 -3962.994} C_VEL
LIN {X 0,Y 538.119,Z 267.758,A -85,B 0,C 180,E1 -3965.997,E2 -3965.997} C_VEL
LIN {X 0,Y 538.067,Z 267.77,A -85,B 0,C 180,E1 -3969.017,E2 -3969.017} C_VEL
LIN {X 0,Y 538.084,Z 267.766,A -85,B 0,C 180,E1 -3972.062,E2 -3972.062} C_VEL
LIN {X 0,Y 538.043,Z 267.78,A -85,B 0,C 180,E1 -3975.143,E2 -3975.143} C_VEL
LIN {X 0,Y 538.026,Z 267.774,A -85,B 0,C 180,E1 -3978.27,E2 -3978.27} C_VEL
LIN {X 0,Y 538.037,Z 267.775,A -85,B 0,C 180,E1 -3980.651,E2 -3980.651} C_VEL
LIN {X 0,Y 538.025,Z 267.775,A -85,B 0,C 180,E1 -3983.887,E2 -3983.887} C_VEL
LIN {X 0,Y 538.041,Z 267.773,A -85,B 0,C 180,E1 -3986.366,E2 -3986.366} C_VEL
LIN {X 0,Y 538.03,Z 267.78,A -85,B 0,C 180,E1 -3988.933,E2 -3988.933} C_VEL
LIN {X 0,Y 538.009,Z 267.776,A -85,B 0,C 180,E1 -3991.887,E2 -3991.887} C_VEL
LIN {X 0,Y 538.026,Z 267.778,A -85,B 0,C 180,E1 -3994.62,E2 -3994.62} C_VEL
LIN {X 0,Y 538.006,Z 267.782,A -85,B 0,C 180,E1 -3997.17,E2 -3997.17} C_VEL
LIN {X 0,Y 538.029,Z 267.773,A -85,B 0,C 180,E1 -3999.796,E2 -3999.796} C_VEL
LIN {X 0,Y 538.019,Z 267.783,A -85,B 0,C 180,E1 -4002.786,E2 -4002.786} C_VEL
LIN {X 0,Y 538.031,Z 267.78,A -85,B 0,C 180,E1 -4005.14,E2 -4005.14} C_VEL
LIN {X 0,Y 538.04,Z 267.773,A -85,B 0,C 180,E1 -4008.228,E2 -4008.228} C_VEL
LIN {X 0,Y 538.014,Z 267.78,A -85,B 0,C 180,E1 -4011.17,E2 -4011.17} C_VEL
LIN {X 0,Y 537.993,Z 267.78,A -85,B 0,C 180,E1 -4014.088,E2 -4014.088} C_VEL
LIN {X 0,Y 538.028,Z 267.78,A -85,B 0,C 180,E1 -4016.727,E2 -4016.727} C_VEL
LIN {X 0,Y 538.025,Z 267.779,A -85,B 0,C 180,E1 -4019.556,E2 -4019.556} C_VEL
LIN {X 0,Y 538.035,Z 267.866,A -85,B 0,C 180,E1 -4020.48,E2 -4020.48} C_VEL
LIN {X 0,Y 542.217,Z 281.883,A -85,B 0,C 180,E1 -4022.051,E2 -4022.051} C_VEL
LIN {X 0,Y 541.836,Z 299.221,A -85,B 0,C 180,E1 -4023.656,E2 -4023.656} C_VEL
LIN {X 0,Y 541.545,Z 311.732,A -85,B 0,C 180,E1 -4024.779,E2 -4024.779} C_VEL
LIN {X 0,Y 543.768,Z 323.454,A -85,B 0,C 180,E1 -4025.056,E2 -4025.056} C_VEL
LIN {X 0,Y 542.504,Z 519.023,A -85,B 0,C 180,E1 -4027.783,E2 -4027.783} C_VEL
LIN {X 0,Y 542.195,Z 534.761,A -85,B 0,C 180,E1 -4028.145,E2 -4028.145} C_VEL
LIN {X 0,Y 541.832,Z 550.675,A -85,B 0,C 180,E1 -4028.654,E2 -4028.654} C_VEL
LIN {X 0,Y 541.423,Z 564.857,A -85,B 0,C 180,E1 -4029.233,E2 -4029.233} C_VEL
LIN {X 0,Y 540.905,Z 580.912,A -85,B 0,C 180,E1 -4030.058,E2 -4030.058} C_VEL
LIN {X 0,Y 540.322,Z 596.22,A -85,B 0,C 180,E1 -4031.024,E2 -4031.024} C_VEL
LIN {X 0,Y 539.828,Z 609.24,A -85,B 0,C 180,E1 -4032.006,E2 -4032.006} C_VEL
LIN {X 0,Y 539.35,Z 622.113,A -85,B 0,C 180,E1 -4033.146,E2 -4033.146} C_VEL
LIN {X 0,Y 538.949,Z 633.284,A -85,B 0,C 180,E1 -4034.301,E2 -4034.301} C_VEL
LIN {X 0,Y 538.586,Z 644.42,A -85,B 0,C 180,E1 -4035.645,E2 -4035.645} C_VEL
LIN {X 0,Y 538.204,Z 655.207,A -85,B 0,C 180,E1 -4037.174,E2 -4037.174} C_VEL
LIN {X 0,Y 537.989,Z 664.267,A -85,B 0,C 180,E1 -4038.7,E2 -4038.7} C_VEL
LIN {X 0,Y 537.739,Z 671.855,A -85,B 0,C 180,E1 -4040.218,E2 -4040.218} C_VEL
LIN {X 0,Y 537.658,Z 679.465,A -85,B 0,C 180,E1 -4042.111,E2 -4042.111} C_VEL
LIN {X 0,Y 537.586,Z 685.249,A -85,B 0,C 180,E1 -4043.997,E2 -4043.997} C_VEL
LIN {X 0,Y 537.5,Z 688.635,A -85,B 0,C 180,E1 -4045.5,E2 -4045.5} C_VEL
LIN {X 0,Y 537.538,Z 691.091,A -85,B 0,C 180,E1 -4047.002,E2 -4047.002} C_VEL
LIN {X 0,Y 537.445,Z 692.479,A -85,B 0,C 180,E1 -4048.501,E2 -4048.501} C_VEL
LIN {X 0,Y 537.437,Z 693,A -85,B 0,C 180,E1 -4050,E2 -4050} C_VEL
LIN {X 0,Y 537.445,Z 692.478,A -85,B 0,C 180,E1 -4051.499,E2 -4051.499} C_VEL
LIN {X 0,Y 537.538,Z 691.089,A -85,B 0,C 180,E1 -4052.998,E2 -4052.998} C_VEL
LIN {X 0,Y 537.5,Z 688.634,A -85,B 0,C 180,E1 -4054.5,E2 -4054.5} C_VEL
LIN {X 0,Y 537.586,Z 685.251,A -85,B 0,C 180,E1 -4056.003,E2 -4056.003} C_VEL
LIN {X 0,Y 537.658,Z 679.467,A -85,B 0,C 180,E1 -4057.889,E2 -4057.889} C_VEL
LIN {X 0,Y 537.739,Z 671.855,A -85,B 0,C 180,E1 -4059.782,E2 -4059.782} C_VEL
LIN {X 0,Y 537.99,Z 664.267,A -85,B 0,C 180,E1 -4061.3,E2 -4061.3} C_VEL
LIN {X 0,Y 538.205,Z 655.207,A -85,B 0,C 180,E1 -4062.826,E2 -4062.826} C_VEL
LIN {X 0,Y 538.585,Z 644.419,A -85,B 0,C 180,E1 -4064.355,E2 -4064.355} C_VEL
LIN {X 0,Y 538.979,Z 633.283,A -85,B 0,C 180,E1 -4065.698,E2 -4065.698} C_VEL
LIN {X 0,Y 539.414,Z 621.135,A -85,B 0,C 180,E1 -4066.949,E2 -4066.949} C_VEL
LIN {X 0,Y 539.949,Z 607.73,A -85,B 0,C 180,E1 -4068.116,E2 -4068.116} C_VEL
LIN {X 0,Y 540.383,Z 594.779,A -85,B 0,C 180,E1 -4069.073,E2 -4069.073} C_VEL
LIN {X 0,Y 540.881,Z 580.892,A -85,B 0,C 180,E1 -4069.943,E2 -4069.943} C_VEL
LIN {X 0,Y 541.402,Z 564.759,A -85,B 0,C 180,E1 -4070.772,E2 -4070.772} C_VEL
LIN {X 0,Y 541.885,Z 549.347,A -85,B 0,C 180,E1 -4071.393,E2 -4071.393} C_VEL
LIN {X 0,Y 542.246,Z 532.895,A -85,B 0,C 180,E1 -4071.903,E2 -4071.903} C_VEL
LIN {X 0,Y 542.497,Z 517.475,A -85,B 0,C 180,E1 -4072.243,E2 -4072.243} C_VEL
LIN {X 0,Y 543.768,Z 323.4,A -85,B 0,C 180,E1 -4074.944,E2 -4074.944} C_VEL
LIN {X 0,Y 541.51,Z 311.069,A -85,B 0,C 180,E1 -4075.255,E2 -4075.255} C_VEL
LIN {X 0,Y 542.344,Z 283.215,A -85,B 0,C 180,E1 -4077.808,E2 -4077.808} C_VEL
LIN {X 0,Y 541.774,Z 280.415,A -85,B 0,C 180,E1 -4078.103,E2 -4078.103} C_VEL
LIN {X 0,Y 538.027,Z 267.783,A -85,B 0,C 180,E1 -4079.533,E2 -4079.533} C_VEL
LIN {X 0,Y 538.018,Z 267.778,A -85,B 0,C 180,E1 -4082.383,E2 -4082.383} C_VEL
LIN {X 0,Y 537.997,Z 267.783,A -85,B 0,C 180,E1 -4085.085,E2 -4085.085} C_VEL
LIN {X 0,Y 537.993,Z 267.781,A -85,B 0,C 180,E1 -4087.878,E2 -4087.878} C_VEL
LIN {X 0,Y 538.051,Z 267.776,A -85,B 0,C 180,E1 -4090.776,E2 -4090.776} C_VEL
LIN {X 0,Y 538.029,Z 267.774,A -85,B 0,C 180,E1 -4094.075,E2 -4094.075} C_VEL
LIN {X 0,Y 538.027,Z 267.783,A -85,B 0,C 180,E1 -4097.013,E2 -4097.013} C_VEL
LIN {X 0,Y 538.052,Z 267.777,A -85,B 0,C 180,E1 -4099.253,E2 -4099.253} C_VEL
LIN {X 0,Y 537.994,Z 267.776,A -85,B 0,C 180,E1 -4102.123,E2 -4102.123} C_VEL
LIN {X 0,Y 537.999,Z 267.786,A -85,B 0,C 180,E1 -4104.916,E2 -4104.916} C_VEL
LIN {X 0,Y 538.019,Z 267.773,A -85,B 0,C 180,E1 -4107.618,E2 -4107.618} C_VEL
LIN {X 0,Y 538.018,Z 267.776,A -85,B 0,C 180,E1 -4110.239,E2 -4110.239} C_VEL
LIN {X 0,Y 538.058,Z 267.771,A -85,B 0,C 180,E1 -4112.796,E2 -4112.796} C_VEL
LIN {X 0,Y 538.05,Z 267.772,A -85,B 0,C 180,E1 -4115.293,E2 -4115.293} C_VEL
LIN {X 0,Y 538.016,Z 267.77,A -85,B 0,C 180,E1 -4118.042,E2 -4118.042} C_VEL
LIN {X 0,Y 538.034,Z 267.777,A -85,B 0,C 180,E1 -4120.94,E2 -4120.94} C_VEL
LIN {X 0,Y 538.016,Z 267.77,A -85,B 0,C 180,E1 -4123.299,E2 -4123.299} C_VEL
LIN {X 0,Y 538.062,Z 267.769,A -85,B 0,C 180,E1 -4125.631,E2 -4125.631} C_VEL
LIN {X 0,Y 538.078,Z 267.766,A -85,B 0,C 180,E1 -4128.702,E2 -4128.702} C_VEL
LIN {X 0,Y 538.061,Z 267.769,A -85,B 0,C 180,E1 -4131.74,E2 -4131.74} C_VEL
LIN {X 0,Y 538.151,Z 267.756,A -85,B 0,C 180,E1 -4134.755,E2 -4134.755} C_VEL
LIN {X 0,Y 538.167,Z 267.755,A -85,B 0,C 180,E1 -4137.755,E2 -4137.755} C_VEL
LIN {X 0,Y 538.18,Z 267.753,A -85,B 0,C 180,E1 -4140.749,E2 -4140.749} C_VEL
LIN {X 0,Y 538.122,Z 267.761,A -85,B 0,C 180,E1 -4142.995,E2 -4142.995} C_VEL
LIN {X 0,Y 538.089,Z 267.77,A -85,B 0,C 180,E1 -4145.998,E2 -4145.998} C_VEL
LIN {X 0,Y 538.049,Z 267.769,A -85,B 0,C 180,E1 -4149.018,E2 -4149.018} C_VEL
LIN {X 0,Y 538.063,Z 267.775,A -85,B 0,C 180,E1 -4152.063,E2 -4152.063} C_VEL
LIN {X 0,Y 538.041,Z 267.77,A -85,B 0,C 180,E1 -4155.144,E2 -4155.144} C_VEL
LIN {X 0,Y 538.005,Z 267.778,A -85,B 0,C 180,E1 -4158.272,E2 -4158.272} C_VEL
LIN {X 0,Y 538.028,Z 267.777,A -85,B 0,C 180,E1 -4160.652,E2 -4160.652} C_VEL
LIN {X 0,Y 538.009,Z 267.778,A -85,B 0,C 180,E1 -4163.878,E2 -4163.878} C_VEL
LIN {X 0,Y 537.976,Z 267.785,A -85,B 0,C 180,E1 -4166.371,E2 -4166.371} C_VEL
LIN {X 0,Y 537.976,Z 267.779,A -85,B 0,C 180,E1 -4168.922,E2 -4168.922} C_VEL
LIN {X 0,Y 537.996,Z 267.782,A -85,B 0,C 180,E1 -4171.884,E2 -4171.884} C_VEL
LIN {X 0,Y 537.991,Z 267.779,A -85,B 0,C 180,E1 -4174.614,E2 -4174.614} C_VEL
LIN {X 0,Y 537.965,Z 267.789,A -85,B 0,C 180,E1 -4177.881,E2 -4177.881} C_VEL
LIN {X 0,Y 537.945,Z 267.786,A -85,B 0,C 180,E1 -4180.253,E2 -4180.253} C_VEL
LIN {X 0,Y 537.279,Z 267.868,A -85,B 0,C 180,E1 -4180.878,E2 -4180.878} C_VEL
LIN {X 0,Y 534.436,Z 268.228,A -85,B 0,C 180,E1 -4181.893,E2 -4181.893} C_VEL
LIN {X 0,Y 532.035,Z 268.53,A -85,B 0,C 180,E1 -4182.71,E2 -4182.71} C_VEL
LIN {X 0,Y 531.005,Z 268.655,A -85,B 0,C 180,E1 -4183.341,E2 -4183.341} C_VEL
LIN {X 0,Y 530.922,Z 268.664,A -85,B 0,C 180,E1 -4183.555,E2 -4183.555} C_VEL
LIN {X 0,Y 530.967,Z 268.657,A -85,B 0,C 180,E1 -4185.624,E2 -4185.624} C_VEL
LIN {X 0,Y 530.913,Z 268.664,A -85,B 0,C 180,E1 -4188.557,E2 -4188.557} C_VEL
LIN {X 0,Y 530.97,Z 268.78,A -85,B 0,C 180,E1 -4189.628,E2 -4189.628} C_VEL
LIN {X 0,Y 534.631,Z 282.059,A -85,B 0,C 180,E1 -4191.287,E2 -4191.287} C_VEL
LIN {X 0,Y 534.783,Z 283.786,A -85,B 0,C 180,E1 -4191.482,E2 -4191.482} C_VEL
LIN {X 0,Y 537.388,Z 296.405,A -85,B 0,C 180,E1 -4191.806,E2 -4191.806} C_VEL
LIN {X 0,Y 535.966,Z 488.876,A -85,B 0,C 180,E1 -4194.527,E2 -4194.527} C_VEL
LIN {X 0,Y 535.597,Z 505.528,A -85,B 0,C 180,E1 -4194.907,E2 -4194.907} C_VEL
LIN {X 0,Y 535.214,Z 522.107,A -85,B 0,C 180,E1 -4195.451,E2 -4195.451} C_VEL
LIN {X 0,Y 534.706,Z 538.283,A -85,B 0,C 180,E1 -4196.148,E2 -4196.148} C_VEL
LIN {X 0,Y 534.168,Z 552.501,A -85,B 0,C 180,E1 -4196.906,E2 -4196.906} C_VEL
LIN {X 0,Y 533.583,Z 567.411,A -85,B 0,C 180,E1 -4197.879,E2 -4197.879} C_VEL
LIN {X 0,Y 533.036,Z 579.987,A -85,B 0,C 180,E1 -4198.857,E2 -4198.857} C_VEL
LIN {X 0,Y 532.416,Z 593.677,A -85,B 0,C 180,E1 -4200.108,E2 -4200.108} C_VEL
LIN {X 0,Y 531.93,Z 605.529,A -85,B 0,C 180,E1 -4201.383,E2 -4201.383} C_VEL
LIN {X 0,Y 531.494,Z 617.153,A -85,B 0,C 180,E1 -4202.858,E2 -4202.858} C_VEL
LIN {X 0,Y 531.157,Z 626.977,A -85,B 0,C 180,E1 -4204.326,E2 -4204.326} C_VEL
LIN {X 0,Y 530.916,Z 635.205,A -85,B 0,C 180,E1 -4205.772,E2 -4205.772} C_VEL
LIN {X 0,Y 530.686,Z 643.064,A -85,B 0,C 180,E1 -4207.415,E2 -4207.415} C_VEL
LIN {X 0,Y 530.539,Z 649.443,A -85,B 0,C 180,E1 -4209.043,E2 -4209.043} C_VEL
LIN {X 0,Y 530.467,Z 654.407,A -85,B 0,C 180,E1 -4210.657,E2 -4210.657} C_VEL
LIN {X 0,Y 530.39,Z 658.784,A -85,B 0,C 180,E1 -4212.564,E2 -4212.564} C_VEL
LIN {X 0,Y 530.331,Z 660.854,A -85,B 0,C 180,E1 -4213.841,E2 -4213.841} C_VEL
LIN {X 0,Y 530.386,Z 662.409,A -85,B 0,C 180,E1 -4215.418,E2 -4215.418} C_VEL
LIN {X 0,Y 530.364,Z 662.993,A -85,B 0,C 180,E1 -4216.981,E2 -4216.981} C_VEL
LIN {X 0,Y 530.452,Z 662.424,A -85,B 0,C 180,E1 -4218.649,E2 -4218.649} C_VEL
LIN {X 0,Y 530.39,Z 661.094,A -85,B 0,C 180,E1 -4220.081,E2 -4220.081} C_VEL
LIN {X 0,Y 530.418,Z 658.606,A -85,B 0,C 180,E1 -4221.619,E2 -4221.619} C_VEL
LIN {X 0,Y 530.52,Z 654.228,A -85,B 0,C 180,E1 -4223.495,E2 -4223.495} C_VEL
LIN {X 0,Y 530.52,Z 649.395,A -85,B 0,C 180,E1 -4225.06,E2 -4225.06} C_VEL
LIN {X 0,Y 530.657,Z 643.45,A -85,B 0,C 180,E1 -4226.583,E2 -4226.583} C_VEL
LIN {X 0,Y 530.848,Z 636.331,A -85,B 0,C 180,E1 -4228.103,E2 -4228.103} C_VEL
LIN {X 0,Y 531.081,Z 627.894,A -85,B 0,C 180,E1 -4229.621,E2 -4229.621} C_VEL
LIN {X 0,Y 531.37,Z 617.837,A -85,B 0,C 180,E1 -4231.137,E2 -4231.137} C_VEL
LIN {X 0,Y 531.874,Z 607.556,A -85,B 0,C 180,E1 -4232.461,E2 -4232.461} C_VEL
LIN {X 0,Y 532.334,Z 595.633,A -85,B 0,C 180,E1 -4233.785,E2 -4233.785} C_VEL
LIN {X 0,Y 532.892,Z 582.623,A -85,B 0,C 180,E1 -4235.012,E2 -4235.012} C_VEL
LIN {X 0,Y 533.463,Z 568.385,A -85,B 0,C 180,E1 -4236.145,E2 -4236.145} C_VEL
LIN {X 0,Y 534.056,Z 554.083,A -85,B 0,C 180,E1 -4237.087,E2 -4237.087} C_VEL
LIN {X 0,Y 534.57,Z 540.379,A -85,B 0,C 180,E1 -4237.84,E2 -4237.84} C_VEL
LIN {X 0,Y 535.111,Z 524.606,A -85,B 0,C 180,E1 -4238.544,E2 -4238.544} C_VEL
LIN {X 0,Y 535.586,Z 508.22,A -85,B 0,C 180,E1 -4239.107,E2 -4239.107} C_VEL
LIN {X 0,Y 535.926,Z 491.821,A -85,B 0,C 180,E1 -4239.506,E2 -4239.506} C_VEL
LIN {X 0,Y 536.202,Z 464.756,A -85,B 0,C 180,E1 -4239.916,E2 -4239.916} C_VEL
LIN {X 0,Y 537.406,Z 296.696,A -85,B 0,C 180,E1 -4242.277,E2 -4242.277} C_VEL
LIN {X 0,Y 534.72,Z 283.61,A -85,B 0,C 180,E1 -4242.62,E2 -4242.62} C_VEL
LIN {X 0,Y 534.393,Z 281.013,A -85,B 0,C 180,E1 -4242.919,E2 -4242.919} C_VEL
LIN {X 0,Y 531.016,Z 268.656,A -85,B 0,C 180,E1 -4244.466,E2 -4244.466} C_VEL
LIN {X 0,Y 530.976,Z 268.655,A -85,B 0,C 180,E1 -4247.724,E2 -4247.724} C_VEL
LIN {X 0,Y 531.017,Z 268.654,A -85,B 0,C 180,E1 -4250.127,E2 -4250.127} C_VEL
LIN {X 0,Y 530.945,Z 268.662,A -85,B 0,C 180,E1 -4252.573,E2 -4252.573} C_VEL
LIN {X 0,Y 530.948,Z 268.656,A -85,B 0,C 180,E1 -4255.06,E2 -4255.06} C_VEL
LIN {X 0,Y 530.952,Z 268.658,A -85,B 0,C 180,E1 -4257.599,E2 -4257.599} C_VEL
LIN {X 0,Y 530.947,Z 268.665,A -85,B 0,C 180,E1 -4260.198,E2 -4260.198} C_VEL
LIN {X 0,Y 530.947,Z 268.657,A -85,B 0,C 180,E1 -4262.868,E2 -4262.868} C_VEL
LIN {X 0,Y 530.92,Z 268.66,A -85,B 0,C 180,E1 -4265.623,E2 -4265.623} C_VEL
LIN {X 0,Y 530.928,Z 268.659,A -85,B 0,C 180,E1 -4268.647,E2 -4268.647} C_VEL
LIN {X 0,Y 530.909,Z 268.662,A -85,B 0,C 180,E1 -4271.444,E2 -4271.444} C_VEL
LIN {X 0,Y 530.96,Z 268.655,A -85,B 0,C 180,E1 -4274.55,E2 -4274.55} C_VEL
LIN {X 0,Y 530.906,Z 268.661,A -85,B 0,C 180,E1 -4277.535,E2 -4277.535} C_VEL
LIN {X 0,Y 530.956,Z 268.653,A -85,B 0,C 180,E1 -4280.553,E2 -4280.553} C_VEL
LIN {X 0,Y 530.905,Z 268.652,A -85,B 0,C 180,E1 -4283.437,E2 -4283.437} C_VEL
LIN {X 0,Y 530.952,Z 268.657,A -85,B 0,C 180,E1 -4286.224,E2 -4286.224} C_VEL
LIN {X 0,Y 530.957,Z 268.657,A -85,B 0,C 180,E1 -4289.358,E2 -4289.358} C_VEL
LIN {X 0,Y 530.952,Z 268.656,A -85,B 0,C 180,E1 -4292.4,E2 -4292.4} C_VEL
LIN {X 0,Y 530.95,Z 268.655,A -85,B 0,C 180,E1 -4294.939,E2 -4294.939} C_VEL
LIN {X 0,Y 530.979,Z 268.657,A -85,B 0,C 180,E1 -4297.898,E2 -4297.898} C_VEL
LIN {X 0,Y 530.983,Z 268.65,A -85,B 0,C 180,E1 -4300.676,E2 -4300.676} C_VEL
LIN {X 0,Y 530.961,Z 268.652,A -85,B 0,C 180,E1 -4303.07,E2 -4303.07} C_VEL
LIN {X 0,Y 531.01,Z 268.655,A -85,B 0,C 180,E1 -4305.435,E2 -4305.435} C_VEL
LIN {X 0,Y 531.036,Z 268.64,A -85,B 0,C 180,E1 -4308.549,E2 -4308.549} C_VEL
LIN {X 0,Y 531.03,Z 268.652,A -85,B 0,C 180,E1 -4311.629,E2 -4311.629} C_VEL
LIN {X 0,Y 531.08,Z 268.637,A -85,B 0,C 180,E1 -4313.922,E2 -4313.922} C_VEL
LIN {X 0,Y 531.093,Z 268.639,A -85,B 0,C 180,E1 -4316.965,E2 -4316.965} C_VEL
LIN {X 0,Y 531.145,Z 268.627,A -85,B 0,C 180,E1 -4320,E2 -4320} C_VEL
LIN {X 0,Y 531.101,Z 268.64,A -85,B 0,C 180,E1 -4323.034,E2 -4323.034} C_VEL
LIN {X 0,Y 531.074,Z 268.635,A -85,B 0,C 180,E1 -4326.077,E2 -4326.077} C_VEL
LIN {X 0,Y 531.055,Z 268.638,A -85,B 0,C 180,E1 -4328.37,E2 -4328.37} C_VEL
LIN {X 0,Y 531.052,Z 268.645,A -85,B 0,C 180,E1 -4331.672,E2 -4331.672} C_VEL
LIN {X 0,Y 531.03,Z 268.651,A -85,B 0,C 180,E1 -4334.955,E2 -4334.955} C_VEL
LIN {X 0,Y 530.981,Z 268.654,A -85,B 0,C 180,E1 -4337.723,E2 -4337.723} C_VEL
LIN {X 0,Y 531.025,Z 268.646,A -85,B 0,C 180,E1 -4340.127,E2 -4340.127} C_VEL
LIN {X 0,Y 530.966,Z 268.659,A -85,B 0,C 180,E1 -4343.396,E2 -4343.396} C_VEL
LIN {X 0,Y 531.013,Z 268.648,A -85,B 0,C 180,E1 -4345.897,E2 -4345.897} C_VEL
LIN {X 0,Y 530.996,Z 268.65,A -85,B 0,C 180,E1 -4348.455,E2 -4348.455} C_VEL
LIN {X 0,Y 530.956,Z 268.663,A -85,B 0,C 180,E1 -4351.079,E2 -4351.079} C_VEL
LIN {X 0,Y 530.988,Z 268.651,A -85,B 0,C 180,E1 -4353.772,E2 -4353.772} C_VEL
LIN {X 0,Y 530.965,Z 268.655,A -85,B 0,C 180,E1 -4356.557,E2 -4356.557} C_VEL
LIN {X 0,Y 530.983,Z 268.651,A -85,B 0,C 180,E1 -4359.854,E2 -4359.854} C_VEL
LIN {X 0,Y 530.979,Z 268.655,A -85,B 0,C 180,E1 -4362.456,E2 -4362.456} C_VEL
LIN {X 0,Y 530.987,Z 268.653,A -85,B 0,C 180,E1 -4365.621,E2 -4365.621} C_VEL
LIN {X 0,Y 530.999,Z 268.654,A -85,B 0,C 180,E1 -4368.565,E2 -4368.565} C_VEL
LIN {X 0,Y 530.957,Z 268.655,A -85,B 0,C 180,E1 -4371.529,E2 -4371.529} C_VEL
LIN {X 0,Y 530.953,Z 268.659,A -85,B 0,C 180,E1 -4374.38,E2 -4374.38} C_VEL
LIN {X 0,Y 530.965,Z 268.659,A -85,B 0,C 180,E1 -4377.133,E2 -4377.133} C_VEL
LIN {X 0,Y 530.989,Z 268.806,A -85,B 0,C 180,E1 -4380.16,E2 -4380.16} C_VEL
LIN {X 0,Y 535.637,Z 284.426,A -85,B 0,C 180,E1 -4381.94,E2 -4381.94} C_VEL
LIN {X 0,Y 534.834,Z 311.103,A -85,B 0,C 180,E1 -4384.424,E2 -4384.424} C_VEL
LIN {X 0,Y 537.276,Z 324.271,A -85,B 0,C 180,E1 -4384.748,E2 -4384.748} C_VEL
LIN {X 0,Y 536.131,Z 502.454,A -85,B 0,C 180,E1 -4387.25,E2 -4387.25} C_VEL
LIN {X 0,Y 535.805,Z 522.278,A -85,B 0,C 180,E1 -4387.566,E2 -4387.566} C_VEL
LIN {X 0,Y 535.524,Z 538.084,A -85,B 0,C 180,E1 -4387.96,E2 -4387.96} C_VEL
LIN {X 0,Y 535.034,Z 555.108,A -85,B 0,C 180,E1 -4388.551,E2 -4388.551} C_VEL
LIN {X 0,Y 534.526,Z 571.66,A -85,B 0,C 180,E1 -4389.307,E2 -4389.307} C_VEL
LIN {X 0,Y 533.952,Z 585.541,A -85,B 0,C 180,E1 -4390.088,E2 -4390.088} C_VEL
LIN {X 0,Y 533.418,Z 600.07,A -85,B 0,C 180,E1 -4391.068,E2 -4391.068} C_VEL
LIN {X 0,Y 532.794,Z 614.125,A -85,B 0,C 180,E1 -4392.194,E2 -4392.194} C_VEL
LIN {X 0,Y 532.246,Z 627.877,A -85,B 0,C 180,E1 -4393.507,E2 -4393.507} C_VEL
LIN {X 0,Y 531.725,Z 640.199,A -85,B 0,C 180,E1 -4394.906,E2 -4394.906} C_VEL
LIN {X 0,Y 531.328,Z 651.403,A -85,B 0,C 180,E1 -4396.421,E2 -4396.421} C_VEL
LIN {X 0,Y 531.036,Z 661.013,A -85,B 0,C 180,E1 -4397.963,E2 -4397.963} C_VEL
LIN {X 0,Y 530.847,Z 668.24,A -85,B 0,C 180,E1 -4399.319,E2 -4399.319} C_VEL
LIN {X 0,Y 530.648,Z 675.099,A -85,B 0,C 180,E1 -4400.855,E2 -4400.855} C_VEL
LIN {X 0,Y 530.553,Z 680.716,A -85,B 0,C 180,E1 -4402.388,E2 -4402.388} C_VEL
LIN {X 0,Y 530.494,Z 685.25,A -85,B 0,C 180,E1 -4403.916,E2 -4403.916} C_VEL
LIN {X 0,Y 530.403,Z 688.634,A -85,B 0,C 180,E1 -4405.44,E2 -4405.44} C_VEL
LIN {X 0,Y 530.443,Z 691.091,A -85,B 0,C 180,E1 -4406.962,E2 -4406.962} C_VEL
LIN {X 0,Y 530.355,Z 692.478,A -85,B 0,C 180,E1 -4408.481,E2 -4408.481} C_VEL
LIN {X 0,Y 530.338,Z 693,A -85,B 0,C 180,E1 -4410,E2 -4410} C_VEL
LIN {X 0,Y 530.355,Z 692.477,A -85,B 0,C 180,E1 -4411.519,E2 -4411.519} C_VEL
LIN {X 0,Y 530.443,Z 691.089,A -85,B 0,C 180,E1 -4413.038,E2 -4413.038} C_VEL
LIN {X 0,Y 530.403,Z 688.633,A -85,B 0,C 180,E1 -4414.56,E2 -4414.56} C_VEL
LIN {X 0,Y 530.494,Z 685.252,A -85,B 0,C 180,E1 -4416.084,E2 -4416.084} C_VEL
LIN {X 0,Y 530.569,Z 679.467,A -85,B 0,C 180,E1 -4417.995,E2 -4417.995} C_VEL
LIN {X 0,Y 530.696,Z 671.855,A -85,B 0,C 180,E1 -4419.913,E2 -4419.913} C_VEL
LIN {X 0,Y 531,Z 663.25,A -85,B 0,C 180,E1 -4421.646,E2 -4421.646} C_VEL
LIN {X 0,Y 531.228,Z 653.974,A -85,B 0,C 180,E1 -4423.192,E2 -4423.192} C_VEL
LIN {X 0,Y 531.634,Z 644.419,A -85,B 0,C 180,E1 -4424.547,E2 -4424.547} C_VEL
LIN {X 0,Y 532.056,Z 633.259,A -85,B 0,C 180,E1 -4425.908,E2 -4425.908} C_VEL
LIN {X 0,Y 532.532,Z 621.019,A -85,B 0,C 180,E1 -4427.175,E2 -4427.175} C_VEL
LIN {X 0,Y 533.095,Z 607.705,A -85,B 0,C 180,E1 -4428.341,E2 -4428.341} C_VEL
LIN {X 0,Y 533.608,Z 594.538,A -85,B 0,C 180,E1 -4429.324,E2 -4429.324} C_VEL
LIN {X 0,Y 534.123,Z 580.645,A -85,B 0,C 180,E1 -4430.206,E2 -4430.206} C_VEL
LIN {X 0,Y 534.714,Z 564.964,A -85,B 0,C 180,E1 -4431.021,E2 -4431.021} C_VEL
LIN {X 0,Y 535.182,Z 550.391,A -85,B 0,C 180,E1 -4431.624,E2 -4431.624} C_VEL
LIN {X 0,Y 535.621,Z 533.538,A -85,B 0,C 180,E1 -4432.163,E2 -4432.163} C_VEL
LIN {X 0,Y 535.906,Z 518.673,A -85,B 0,C 180,E1 -4432.506,E2 -4432.506} C_VEL
LIN {X 0,Y 537.169,Z 344.104,A -85,B 0,C 180,E1 -4434.969,E2 -4434.969} C_VEL
LIN {X 0,Y 537.181,Z 323.803,A -85,B 0,C 180,E1 -4435.262,E2 -4435.262} C_VEL
LIN {X 0,Y 534.82,Z 310.939,A -85,B 0,C 180,E1 -4435.585,E2 -4435.585} C_VEL
LIN {X 0,Y 535.645,Z 284.381,A -85,B 0,C 180,E1 -4438.055,E2 -4438.055} C_VEL
LIN {X 0,Y 530.981,Z 268.659,A -85,B 0,C 180,E1 -4439.868,E2 -4439.868} C_VEL
LIN {X 0,Y 530.966,Z 268.658,A -85,B 0,C 180,E1 -4442.867,E2 -4442.867} C_VEL
LIN {X 0,Y 530.953,Z 268.66,A -85,B 0,C 180,E1 -4445.62,E2 -4445.62} C_VEL
LIN {X 0,Y 530.968,Z 268.658,A -85,B 0,C 180,E1 -4448.654,E2 -4448.654} C_VEL
LIN {X 0,Y 530.999,Z 268.651,A -85,B 0,C 180,E1 -4451.435,E2 -4451.435} C_VEL
LIN {X 0,Y 530.989,Z 268.653,A -85,B 0,C 180,E1 -4454.547,E2 -4454.547} C_VEL
LIN {X 0,Y 530.988,Z 268.649,A -85,B 0,C 180,E1 -4457.834,E2 -4457.834} C_VEL
LIN {X 0,Y 530.991,Z 268.654,A -85,B 0,C 180,E1 -4460.557,E2 -4460.557} C_VEL
LIN {X 0,Y 530.955,Z 268.657,A -85,B 0,C 180,E1 -4463.442,E2 -4463.442} C_VEL
LIN {X 0,Y 530.999,Z 268.651,A -85,B 0,C 180,E1 -4466.495,E2 -4466.495} C_VEL
LIN {X 0,Y 530.975,Z 268.655,A -85,B 0,C 180,E1 -4469.355,E2 -4469.355} C_VEL
LIN {X 0,Y 531.013,Z 268.643,A -85,B 0,C 180,E1 -4472.468,E2 -4472.468} C_VEL
LIN {X 0,Y 531.007,Z 268.654,A -85,B 0,C 180,E1 -4474.943,E2 -4474.943} C_VEL
LIN {X 0,Y 530.973,Z 268.648,A -85,B 0,C 180,E1 -4478.247,E2 -4478.247} C_VEL
LIN {X 0,Y 530.994,Z 268.659,A -85,B 0,C 180,E1 -4480.678,E2 -4480.678} C_VEL
LIN {X 0,Y 530.981,Z 268.648,A -85,B 0,C 180,E1 -4483.071,E2 -4483.071} C_VEL
LIN {X 0,Y 531.018,Z 268.647,A -85,B 0,C 180,E1 -4485.436,E2 -4485.436} C_VEL
LIN {X 0,Y 531.036,Z 268.645,A -85,B 0,C 180,E1 -4488.55,E2 -4488.55} C_VEL
LIN {X 0,Y 531.036,Z 268.644,A -85,B 0,C 180,E1 -4491.63,E2 -4491.63} C_VEL
LIN {X 0,Y 531.109,Z 268.633,A -85,B 0,C 180,E1 -4494.686,E2 -4494.686} C_VEL
LIN {X 0,Y 531.139,Z 268.631,A -85,B 0,C 180,E1 -4497.725,E2 -4497.725} C_VEL
LIN {X 0,Y 531.15,Z 268.628,A -85,B 0,C 180,E1 -4500.759,E2 -4500.759} C_VEL
LIN {X 0,Y 531.063,Z 268.64,A -85,B 0,C 180,E1 -4503.035,E2 -4503.035} C_VEL
LIN {X 0,Y 531.048,Z 268.648,A -85,B 0,C 180,E1 -4506.078,E2 -4506.078} C_VEL
LIN {X 0,Y 531.011,Z 268.645,A -85,B 0,C 180,E1 -4509.139,E2 -4509.139} C_VEL
LIN {X 0,Y 531.052,Z 268.644,A -85,B 0,C 180,E1 -4511.671,E2 -4511.671} C_VEL
LIN {X 0,Y 531.026,Z 268.645,A -85,B 0,C 180,E1 -4514.953,E2 -4514.953} C_VEL
LIN {X 0,Y 530.974,Z 268.655,A -85,B 0,C 180,E1 -4517.724,E2 -4517.724} C_VEL
LIN {X 0,Y 531.016,Z 268.649,A -85,B 0,C 180,E1 -4520.128,E2 -4520.128} C_VEL
LIN {X 0,Y 530.935,Z 268.658,A -85,B 0,C 180,E1 -4522.574,E2 -4522.574} C_VEL
LIN {X 0,Y 530.941,Z 268.656,A -85,B 0,C 180,E1 -4525.061,E2 -4525.061} C_VEL
LIN {X 0,Y 530.951,Z 268.657,A -85,B 0,C 180,E1 -4527.6,E2 -4527.6} C_VEL
LIN {X 0,Y 530.945,Z 268.658,A -85,B 0,C 180,E1 -4530.639,E2 -4530.639} C_VEL
LIN {X 0,Y 530.948,Z 268.658,A -85,B 0,C 180,E1 -4533.497,E2 -4533.497} C_VEL
LIN {X 0,Y 530.891,Z 268.67,A -85,B 0,C 180,E1 -4536.145,E2 -4536.145} C_VEL
LIN {X 0,Y 530.94,Z 268.658,A -85,B 0,C 180,E1 -4538.65,E2 -4538.65} C_VEL
LIN {X 0,Y 530.91,Z 268.663,A -85,B 0,C 180,E1 -4541.444,E2 -4541.444} C_VEL
LIN {X 0,Y 530.922,Z 268.664,A -85,B 0,C 180,E1 -4543.555,E2 -4543.555} C_VEL
LIN {X 0,Y 530.26,Z 268.747,A -85,B 0,C 180,E1 -4544.189,E2 -4544.189} C_VEL
LIN {X 0,Y 527.423,Z 269.098,A -85,B 0,C 180,E1 -4545.218,E2 -4545.218} C_VEL
LIN {X 0,Y 525.015,Z 269.401,A -85,B 0,C 180,E1 -4546.047,E2 -4546.047} C_VEL
LIN {X 0,Y 523.969,Z 269.527,A -85,B 0,C 180,E1 -4546.686,E2 -4546.686} C_VEL
LIN {X 0,Y 523.878,Z 269.537,A -85,B 0,C 180,E1 -4546.903,E2 -4546.903} C_VEL
LIN {X 0,Y 523.917,Z 269.675,A -85,B 0,C 180,E1 -4549.301,E2 -4549.301} C_VEL
LIN {X 0,Y 528.027,Z 284.287,A -85,B 0,C 180,E1 -4551.141,E2 -4551.141} C_VEL
LIN {X 0,Y 530.99,Z 297.709,A -85,B 0,C 180,E1 -4551.496,E2 -4551.496} C_VEL
LIN {X 0,Y 529.413,Z 489.082,A -85,B 0,C 180,E1 -4554.234,E2 -4554.234} C_VEL
LIN {X 0,Y 529.038,Z 505.439,A -85,B 0,C 180,E1 -4554.611,E2 -4554.611} C_VEL
LIN {X 0,Y 528.623,Z 521.37,A -85,B 0,C 180,E1 -4555.132,E2 -4555.132} C_VEL
LIN {X 0,Y 528.159,Z 536.25,A -85,B 0,C 180,E1 -4555.762,E2 -4555.762} C_VEL
LIN {X 0,Y 527.56,Z 551.144,A -85,B 0,C 180,E1 -4556.551,E2 -4556.551} C_VEL
LIN {X 0,Y 526.932,Z 565.714,A -85,B 0,C 180,E1 -4557.493,E2 -4557.493} C_VEL
LIN {X 0,Y 526.307,Z 578.873,A -85,B 0,C 180,E1 -4558.503,E2 -4558.503} C_VEL
LIN {X 0,Y 525.68,Z 591.992,A -85,B 0,C 180,E1 -4559.689,E2 -4559.689} C_VEL
LIN {X 0,Y 525.133,Z 604.077,A -85,B 0,C 180,E1 -4560.978,E2 -4560.978} C_VEL
LIN {X 0,Y 524.679,Z 614.053,A -85,B 0,C 180,E1 -4562.222,E2 -4562.222} C_VEL
LIN {X 0,Y 524.228,Z 624.544,A -85,B 0,C 180,E1 -4563.742,E2 -4563.742} C_VEL
LIN {X 0,Y 523.942,Z 633.199,A -85,B 0,C 180,E1 -4565.217,E2 -4565.217} C_VEL
LIN {X 0,Y 523.689,Z 640.378,A -85,B 0,C 180,E1 -4566.678,E2 -4566.678} C_VEL
LIN {X 0,Y 523.521,Z 647.251,A -85,B 0,C 180,E1 -4568.335,E2 -4568.335} C_VEL
LIN {X 0,Y 523.462,Z 652.898,A -85,B 0,C 180,E1 -4570.023,E2 -4570.023} C_VEL
LIN {X 0,Y 523.299,Z 657.851,A -85,B 0,C 180,E1 -4572.007,E2 -4572.007} C_VEL
LIN {X 0,Y 523.236,Z 660.59,A -85,B 0,C 180,E1 -4573.616,E2 -4573.616} C_VEL
LIN {X 0,Y 523.277,Z 662.315,A -85,B 0,C 180,E1 -4575.245,E2 -4575.245} C_VEL
LIN {X 0,Y 523.263,Z 662.956,A -85,B 0,C 180,E1 -4576.801,E2 -4576.801} C_VEL
LIN {X 0,Y 523.366,Z 662.465,A -85,B 0,C 180,E1 -4578.604,E2 -4578.604} C_VEL
LIN {X 0,Y 523.31,Z 661.283,A -85,B 0,C 180,E1 -4579.945,E2 -4579.945} C_VEL
LIN {X 0,Y 523.304,Z 658.939,A -85,B 0,C 180,E1 -4581.504,E2 -4581.504} C_VEL
LIN {X 0,Y 523.372,Z 655.626,A -85,B 0,C 180,E1 -4583.058,E2 -4583.058} C_VEL
LIN {X 0,Y 523.469,Z 651.206,A -85,B 0,C 180,E1 -4584.607,E2 -4584.607} C_VEL
LIN {X 0,Y 523.555,Z 645.774,A -85,B 0,C 180,E1 -4586.151,E2 -4586.151} C_VEL
LIN {X 0,Y 523.778,Z 637.269,A -85,B 0,C 180,E1 -4588.078,E2 -4588.078} C_VEL
LIN {X 0,Y 524.057,Z 629.009,A -85,B 0,C 180,E1 -4589.616,E2 -4589.616} C_VEL
LIN {X 0,Y 524.372,Z 619.224,A -85,B 0,C 180,E1 -4591.152,E2 -4591.152} C_VEL
LIN {X 0,Y 524.892,Z 609.189,A -85,B 0,C 180,E1 -4592.494,E2 -4592.494} C_VEL
LIN {X 0,Y 525.43,Z 597.532,A -85,B 0,C 180,E1 -4593.835,E2 -4593.835} C_VEL
LIN {X 0,Y 526.06,Z 583.729,A -85,B 0,C 180,E1 -4595.174,E2 -4595.174} C_VEL
LIN {X 0,Y 526.673,Z 569.597,A -85,B 0,C 180,E1 -4596.32,E2 -4596.32} C_VEL
LIN {X 0,Y 527.278,Z 555.516,A -85,B 0,C 180,E1 -4597.274,E2 -4597.274} C_VEL
LIN {X 0,Y 527.922,Z 540.206,A -85,B 0,C 180,E1 -4598.131,E2 -4598.131} C_VEL
LIN {X 0,Y 528.506,Z 524.31,A -85,B 0,C 180,E1 -4598.845,E2 -4598.845} C_VEL
LIN {X 0,Y 529.01,Z 508.571,A -85,B 0,C 180,E1 -4599.39,E2 -4599.39} C_VEL
LIN {X 0,Y 529.386,Z 492.199,A -85,B 0,C 180,E1 -4599.793,E2 -4599.793} C_VEL
LIN {X 0,Y 529.625,Z 467.368,A -85,B 0,C 180,E1 -4600.18,E2 -4600.18} C_VEL
LIN {X 0,Y 530.982,Z 298.271,A -85,B 0,C 180,E1 -4602.584,E2 -4602.584} C_VEL
LIN {X 0,Y 528.052,Z 284.309,A -85,B 0,C 180,E1 -4602.945,E2 -4602.945} C_VEL
LIN {X 0,Y 523.987,Z 269.53,A -85,B 0,C 180,E1 -4604.803,E2 -4604.803} C_VEL
LIN {X 0,Y 523.919,Z 269.538,A -85,B 0,C 180,E1 -4607.971,E2 -4607.971} C_VEL
LIN {X 0,Y 523.953,Z 269.535,A -85,B 0,C 180,E1 -4610.411,E2 -4610.411} C_VEL
LIN {X 0,Y 523.911,Z 269.536,A -85,B 0,C 180,E1 -4612.893,E2 -4612.893} C_VEL
LIN {X 0,Y 523.885,Z 269.536,A -85,B 0,C 180,E1 -4615.422,E2 -4615.422} C_VEL
LIN {X 0,Y 523.898,Z 269.542,A -85,B 0,C 180,E1 -4618.003,E2 -4618.003} C_VEL
LIN {X 0,Y 523.906,Z 269.535,A -85,B 0,C 180,E1 -4620.846,E2 -4620.846} C_VEL
LIN {X 0,Y 523.914,Z 269.536,A -85,B 0,C 180,E1 -4623.726,E2 -4623.726} C_VEL
LIN {X 0,Y 523.847,Z 269.545,A -85,B 0,C 180,E1 -4626.392,E2 -4626.392} C_VEL
LIN {X 0,Y 523.887,Z 269.534,A -85,B 0,C 180,E1 -4629.088,E2 -4629.088} C_VEL
LIN {X 0,Y 523.887,Z 269.54,A -85,B 0,C 180,E1 -4632.125,E2 -4632.125} C_VEL
LIN {X 0,Y 523.931,Z 269.531,A -85,B 0,C 180,E1 -4635.311,E2 -4635.311} C_VEL
LIN {X 0,Y 523.88,Z 269.537,A -85,B 0,C 180,E1 -4638.699,E2 -4638.699} C_VEL
LIN {X 0,Y 523.899,Z 269.529,A -85,B 0,C 180,E1 -4641.896,E2 -4641.896} C_VEL
LIN {X 0,Y 523.914,Z 269.523,A -85,B 0,C 180,E1 -4644.913,E2 -4644.913} C_VEL
LIN {X 0,Y 523.931,Z 269.536,A -85,B 0,C 180,E1 -4647.681,E2 -4647.681} C_VEL
LIN {X 0,Y 523.936,Z 269.524,A -85,B 0,C 180,E1 -4650.68,E2 -4650.68} C_VEL
LIN {X 0,Y 523.899,Z 269.542,A -85,B 0,C 180,E1 -4653.724,E2 -4653.724} C_VEL
LIN {X 0,Y 523.91,Z 269.53,A -85,B 0,C 180,E1 -4656.269,E2 -4656.269} C_VEL
LIN {X 0,Y 523.947,Z 269.528,A -85,B 0,C 180,E1 -4658.766,E2 -4658.766} C_VEL
LIN {X 0,Y 523.938,Z 269.531,A -85,B 0,C 180,E1 -4661.22,E2 -4661.22} C_VEL
LIN {X 0,Y 523.918,Z 269.537,A -85,B 0,C 180,E1 -4663.638,E2 -4663.638} C_VEL
LIN {X 0,Y 523.927,Z 269.532,A -85,B 0,C 180,E1 -4666.027,E2 -4666.027} C_VEL
LIN {X 0,Y 524.015,Z 269.515,A -85,B 0,C 180,E1 -4668.394,E2 -4668.394} C_VEL
LIN {X 0,Y 523.983,Z 269.532,A -85,B 0,C 180,E1 -4671.515,E2 -4671.515} C_VEL
LIN {X 0,Y 524.043,Z 269.514,A -85,B 0,C 180,E1 -4673.841,E2 -4673.841} C_VEL
LIN {X 0,Y 524.034,Z 269.518,A -85,B 0,C 180,E1 -4676.924,E2 -4676.924} C_VEL
LIN {X 0,Y 524.115,Z 269.502,A -85,B 0,C 180,E1 -4680,E2 -4680} C_VEL
LIN {X 0,Y 524.068,Z 269.517,A -85,B 0,C 180,E1 -4683.075,E2 -4683.075} C_VEL
LIN {X 0,Y 524.033,Z 269.511,A -85,B 0,C 180,E1 -4686.159,E2 -4686.159} C_VEL
LIN {X 0,Y 524.004,Z 269.517,A -85,B 0,C 180,E1 -4688.484,E2 -4688.484} C_VEL
LIN {X 0,Y 524.003,Z 269.522,A -85,B 0,C 180,E1 -4691.739,E2 -4691.739} C_VEL
LIN {X 0,Y 523.992,Z 269.529,A -85,B 0,C 180,E1 -4695.051,E2 -4695.051} C_VEL
LIN {X 0,Y 523.947,Z 269.528,A -85,B 0,C 180,E1 -4697.969,E2 -4697.969} C_VEL
LIN {X 0,Y 523.972,Z 269.526,A -85,B 0,C 180,E1 -4700.41,E2 -4700.41} C_VEL
LIN {X 0,Y 523.917,Z 269.536,A -85,B 0,C 180,E1 -4702.893,E2 -4702.893} C_VEL
LIN {X 0,Y 523.953,Z 269.532,A -85,B 0,C 180,E1 -4705.418,E2 -4705.418} C_VEL
LIN {X 0,Y 523.967,Z 269.524,A -85,B 0,C 180,E1 -4707.999,E2 -4707.999} C_VEL
LIN {X 0,Y 523.944,Z 269.535,A -85,B 0,C 180,E1 -4710.854,E2 -4710.854} C_VEL
LIN {X 0,Y 523.96,Z 269.527,A -85,B 0,C 180,E1 -4713.734,E2 -4713.734} C_VEL
LIN {X 0,Y 523.919,Z 269.531,A -85,B 0,C 180,E1 -4716.404,E2 -4716.404} C_VEL
LIN {X 0,Y 523.923,Z 269.537,A -85,B 0,C 180,E1 -4719.084,E2 -4719.084} C_VEL
LIN {X 0,Y 523.955,Z 269.528,A -85,B 0,C 180,E1 -4722.118,E2 -4722.118} C_VEL
LIN {X 0,Y 523.955,Z 269.531,A -85,B 0,C 180,E1 -4725.308,E2 -4725.308} C_VEL
LIN {X 0,Y 523.961,Z 269.533,A -85,B 0,C 180,E1 -4728.689,E2 -4728.689} C_VEL
LIN {X 0,Y 523.915,Z 269.532,A -85,B 0,C 180,E1 -4731.898,E2 -4731.898} C_VEL
LIN {X 0,Y 523.923,Z 269.537,A -85,B 0,C 180,E1 -4734.911,E2 -4734.911} C_VEL
LIN {X 0,Y 523.933,Z 269.533,A -85,B 0,C 180,E1 -4737.68,E2 -4737.68} C_VEL
LIN {X 0,Y 523.959,Z 269.683,A -85,B 0,C 180,E1 -4739.829,E2 -4739.829} C_VEL
LIN {X 0,Y 529.052,Z 287.016,A -85,B 0,C 180,E1 -4741.829,E2 -4741.829} C_VEL
LIN {X 0,Y 528.167,Z 311.001,A -85,B 0,C 180,E1 -4744.087,E2 -4744.087} C_VEL
LIN {X 0,Y 530.875,Z 326.343,A -85,B 0,C 180,E1 -4744.455,E2 -4744.455} C_VEL
LIN {X 0,Y 529.366,Z 516.952,A -85,B 0,C 180,E1 -4747.175,E2 -4747.175} C_VEL
LIN {X 0,Y 529.037,Z 533.336,A -85,B 0,C 180,E1 -4747.547,E2 -4747.547} C_VEL
LIN {X 0,Y 528.542,Z 550.195,A -85,B 0,C 180,E1 -4748.09,E2 -4748.09} C_VEL
LIN {X 0,Y 528.015,Z 565.868,A -85,B 0,C 180,E1 -4748.755,E2 -4748.755} C_VEL
LIN {X 0,Y 527.406,Z 580.452,A -85,B 0,C 180,E1 -4749.525,E2 -4749.525} C_VEL
LIN {X 0,Y 526.76,Z 595.771,A -85,B 0,C 180,E1 -4750.516,E2 -4750.516} C_VEL
LIN {X 0,Y 526.186,Z 608.522,A -85,B 0,C 180,E1 -4751.497,E2 -4751.497} C_VEL
LIN {X 0,Y 525.602,Z 621.792,A -85,B 0,C 180,E1 -4752.692,E2 -4752.692} C_VEL
LIN {X 0,Y 525.098,Z 633.044,A -85,B 0,C 180,E1 -4753.876,E2 -4753.876} C_VEL
LIN {X 0,Y 524.654,Z 644.271,A -85,B 0,C 180,E1 -4755.255,E2 -4755.255} C_VEL
